(* CoDeSys 2.3.9.55 project: coolingskidlogic.pro *)
(* Libraries: Standard.lib 20.5.14 01:13:26, Iecsfc.lib 30.1.13 06:05:12, SYSLIBCALLBACK.LIB 30.1.13 06:05:12 *)

(* PLC configuration (modules and I/O channels)
xWaterLow AT %IX10.0 [BOOLOnX_I] Ch_1 Digital input
xWaterLowLow AT %IX10.1 [BOOLOnX_I] Ch_2 Digital input
AT %IX10.2 [BOOLOnX_I] Ch_1 Digital input
AT %IX10.3 [BOOLOnX_I] Ch_2 Digital input
AT %IX10.4 [BOOLOnX_I] Ch_3 Digital input
AT %IX10.5 [BOOLOnX_I] Ch_4 Digital input
0750-0402 4 DI 24 V DC 3.0ms [Type_1_4_Channels] node 2, in %IX10.2 out %QB4
  AT %IX10.6 [BOOLOnX_I] Ch_1 Digital input
  AT %IX10.7 [BOOLOnX_I] Ch_2 Digital input
  AT %IX10.8 [BOOLOnX_I] Ch_3 Digital input
  AT %IX10.9 [BOOLOnX_I] Ch_4 Digital input
xOutput8DO1 AT %QX2.0 [BOOLOnX_Q] Ch_1 Digital output
AT %QX2.1 [BOOLOnX_Q] Ch_2 Digital output
AT %QX2.2 [BOOLOnX_Q] Ch_3 Digital output
AT %QX2.3 [BOOLOnX_Q] Ch_4 Digital output
AT %QX2.4 [BOOLOnX_Q] Ch_5 Digital output
AT %QX2.5 [BOOLOnX_Q] Ch_6 Digital output
AT %QX2.6 [BOOLOnX_Q] Ch_7 Digital output
AT %QX2.7 [BOOLOnX_Q] Ch_8 Digital output
xOutput AT %QX2.8 [BOOLOnX_Q] Ch_1 Digital output
AT %QX2.9 [BOOLOnX_Q] Ch_2 Digital output
AT %QX2.10 [BOOLOnX_Q] Ch_1 Digital output
AT %QX2.11 [BOOLOnX_Q] Ch_2 Digital output
0750-0492 2 AI 4-20mA Diff Measurement Input [Type_8_2_Channels] node 6, in %IB20 out %QB0
  AT %IW0 [WORDOnW_I] Ch_1 Input word
  AT %IW1 [WORDOnW_I] Ch_2 Input word
0750-0461 2 AI PT100 (RTD) [Type_44_2_Channels] node 7, in %IB20 out %QB0
  AT %IW2 [INTOnW_I] Ch_1 signed Input value
  AT %IW3 [INTOnW_I] Ch_2 signed Input value
0750-0461 2 AI PT100 (RTD) [Type_44_2_Channels] node 8, in %IB24 out %QB0
  AT %IW4 [INTOnW_I] Ch_1 signed Input value
  AT %IW5 [INTOnW_I] Ch_2 signed Input value
0750-0455 4 AI 4-20mA s.e. [Type_8_4_Channels] node 9, in %IB28 out %QB0
  AT %IW6 [WORDOnW_I] Ch_1 Input word
  AT %IW7 [WORDOnW_I] Ch_2 Input word
  AT %IW8 [WORDOnW_I] Ch_3 Input word
  AT %IW9 [WORDOnW_I] Ch_4 Input word
0750-0554 2 AO 4-20mA [Type_14_2_Channels] node 10, in %IB32 out %QB0
  AT %QW0 [WORDOnW_Q] Ch_1 Analog output
  AT %QW1 [WORDOnW_Q] Ch_2 Analog output
AT %IX10.10 [BOOLOnX_I] Ch_1 Digital input
AT %IX10.11 [BOOLOnX_I] Ch_2 Digital input
AT %IX10.12 [BOOLOnX_I] Ch_3 Digital input
AT %IX10.13 [BOOLOnX_I] Ch_4 Digital input
Modbus variables [PFC200MODBUS] node 1, in %IB0 out %QB0 {PlcStopBehaviour = 1; FiledbusErrorBehaviour = 1; TcpOperation = 1; TcpPort = 502; TcpTimeout = 600; UdpOperation = 1; UdpPort = 502; RtuOperation = 0; NodeId = 1; ResponseTimeout = 100; Interface = 0; Baud = 115200; StopBits = 1; Parity = 1; FlowCtrl = 0; PhysInterface = 0}
Modbus-Master [MB_MASTER] node 2, in %IB0 out %QB0
*)

(* Global variable list: Global_Variables *)
VAR_GLOBAL
	gaPumps: ARRAY [1..2] OF  ST_PUMP;
	gaTemps: ARRAY [1..3] OF ST_RTD;
	gaSwitches: ARRAY [1..3] OF ST_SWITCH;
	gaFans: ARRAY [1..4] OF ST_FAN;
	gConductivity: ST_COND;
	gFlow: ST_FLOW;
	gAct: ST_ACT;
	gSystem: ST_SYSTEM;
	gcAlarm: INT :=  1;
	gcFault:  INT := 0;
	gTempValCtrlSys: ST_TempValCtrlSys;
	gProgramErrors: ST_ProgramErrors;
	tbFailure: BOOL;
	tbSuccess: BOOL;
	tbTBLog: STRING(256);

	activePump: ST_PUMP;
	standbyPump: ST_PUMP;


END_VAR

(* Data type in Legacy *)
TYPE BAD :
STRUCT
END_STRUCT
END_TYPE

(* Data type in Legacy *)
TYPE HERE :
STRUCT
	On: BOOL;
	Off: BOOL;
	Fault: BOOL;
	Shutting_Down: BOOL;
	Initializing: BOOL;
	Calibrating: BOOL;
	Acknowledge_Fault: BOOL;
	LIST_FLAGS: ARRAY [1..25] OF BOOL;
	System_Active: BOOL;
	ManualRequest: BOOL;
	AutoRequest: BOOL;
	BAD_Duplex: BOOL;
	ALERT_Simplex: BOOL;
	REQ_Switch: BOOL;
	ALERT_PriActive: BOOL;
	ALERT_SecActive: BOOL;
END_STRUCT
END_TYPE

(* Data type in Instrument Data Types *)
TYPE RAWINPUT :
STRUCT
	wRawAnalogWord: WORD;
	iRawAnalogInt: INT;
	xRawDigital: BOOL;
END_STRUCT
END_TYPE

(* Data type in Legacy *)
TYPE SignalIO :
STRUCT
END_STRUCT
END_TYPE

(* Data type in Legacy *)
TYPE ST_ACT :
STRUCT
	stDescription: ST_Description;
	stActualization: ST_Analog;
	stCounters: ST_LGCount;
	stCalibrationStatus: ST_CalTest;
	rOpenPerc: REAL; (*Percentage of it being Open*)
END_STRUCT
END_TYPE

(* Data type in Legacy *)
TYPE ST_ActivePumpStandbyPump :
STRUCT
END_STRUCT
END_TYPE

(* Data type in Legacy *)
TYPE ST_Analog :
STRUCT
	rGain: REAL;
	rOffset: REAL;
	iRaw: REAL;
	rProcessed: REAL;
END_STRUCT
END_TYPE

(* Data type in Legacy *)
TYPE ST_Backup :
STRUCT
	xActive: BOOL;
	xRedundant: BOOL;
END_STRUCT
END_TYPE

(* Data type in Legacy *)
TYPE ST_CalTest :
STRUCT
	xCalibrated: BOOL;
	xTested: BOOL;
END_STRUCT
END_TYPE

(* Data type in Legacy *)
TYPE ST_COND :
STRUCT
	stDescription: ST_Description;
	stConductivity: ST_Analog; (*Cond Reading Power*)
	stFault: ST_Digital; (*Fault Y/N*)
	stAlarm: ST_DIgital; (*Alarm Y/N*)
	stCounters: ST_LGCount;
	stCalibrationStatus: ST_CalTest;
END_STRUCT
END_TYPE

(* Data type in Legacy *)
TYPE ST_Count :
STRUCT
	iAlarm: INT;
	iFault: INT;
	iForce: INT;
	iCalibrate: INT;
	iTest: INT;
END_STRUCT
END_TYPE

(* Data type in Instrument Data Types *)
TYPE ST_DC :
STRUCT
	arRealValues: ARRAY [1..10] OF REAL;
	axBoolValues: ARRAY [1..10] OF BOOL;
	aiIntValues: ARRAY [1..10] OF INT;
	awWordValues: ARRAY [1..10] OF WORD;
END_STRUCT
END_TYPE

(* Data type in Legacy *)
TYPE ST_Description :
STRUCT
	iID : INT;
	iState: INT; (*Offline, Standby,  Active, Calibration, Testing *)
	xFault: BOOL;
	xAlarm: BOOL;
	sDetail:  STRING;
END_STRUCT
END_TYPE

(* Data type in Legacy *)
TYPE ST_Digital :
STRUCT
	iValue: INT;
END_STRUCT
END_TYPE

(* Data type in Legacy *)
TYPE ST_FA :
STRUCT
	xFault: BOOL;
	xAlarm: BOOL;
END_STRUCT
END_TYPE

(* Data type in Legacy *)
TYPE ST_FAN :
STRUCT
	stDescription: ST_Description;
	stActivate: ST_Digital; (*Pump On/Off*)
	stCounters: ST_LGCount;
	stCalibrationStatus: ST_CalTest;
	stBackup: ST_Backup;
END_STRUCT
END_TYPE

(* Data type in Legacy *)
TYPE ST_FLOW :
STRUCT
	stDescription: ST_Description;
	stFlowRate: ST_Analog; (*Switch Trip*)
	stCounters: ST_LGCount;
	stCalibrationStatus: ST_CalTest;
END_STRUCT
END_TYPE

(* Data type in Legacy *)
TYPE ST_HeartBeat :
STRUCT
	stDescription: ST_Description;
END_STRUCT
END_TYPE

(* Data type in Instrument Data Types *)
TYPE ST_INSTRUMENT :
STRUCT
	iState: INT; (*0 = Standby; 1 = Data Loading;*)
	stInput: ST_IO;
	stOutput: ST_IO;
	stMeasurement: ST_MEASUREMENTS;
	stActuateValues: ST_MEASUREMENTS;
END_STRUCT
END_TYPE

(* Data type in Flags *)
TYPE ST_InstrumentFlags :
STRUCT
	xConductivitySensorAlarmTrip: BOOL := FALSE;
	xConductivitySensorFaultTrip: BOOL := FALSE;
	xPump1BadRead: BOOL := FALSE;
	xPump2BadRead: BOOL := FALSE;
	xPump1LPError: BOOL := FALSE;
	xPump2LPError: BOOL := FALSE;
	xConductivitySensorBadRead: BOOL := FALSE;
	xConductivitySensorMisalignment: BOOL := FALSE;
	xConductivitySensorError: BOOL := FALSE;
	xFlowSensorBadRead: BOOL := FALSE;
	xRTD1BadRead: BOOL := FALSE;
	xRTD2BadRead: BOOL := FALSE;
	xRTD3BadRead: BOOL := FALSE;
	xNoPumpBackup: BOOL := FALSE;
	xPump1Failure: BOOL := FALSE;
	xPump2Failure: BOOL := FALSE;
	xRTD1Failure: BOOL := FALSE;
	xRTD2Failure: BOOL := FALSE;
	xRTD3Failure: BOOL := FALSE;
	xConductivitySensorFailure: BOOL := FALSE;
	xFlowSensorFailure: BOOL := FALSE;
	xPressureLow: BOOL := FALSE;
	xPumpPowerLow: BOOL := FALSE;
	xFlowLow: BOOL := FALSE;
	xWaterLevelSensorError: BOOL := FALSE;
END_STRUCT
END_TYPE

(* Data type in Legacy *)
TYPE ST_IO :
STRUCT
	axDigital: ARRAY [1..100] OF BOOL;
	awAnalog: ARRAY[1..100] OF WORD;
	aiAnalog: ARRAY[1..100] OF INT;
END_STRUCT
END_TYPE

(* Data type in Legacy *)
TYPE ST_LGCount :
STRUCT
	stLocal : ST_Count;
	stGlobal: ST_Count;
END_STRUCT
END_TYPE

(* Data type in Instrument Data Types *)
TYPE ST_MEASUREMENTS :
STRUCT
	axDigital: ARRAY [1..100] OF BOOL;
	arAnalog: ARRAY[1..100] OF REAL;
END_STRUCT
END_TYPE

(* Data type in Legacy *)
TYPE ST_PRES :
STRUCT
	stDescription: ST_Description;
	stSwitchTrip: ST_Digital; (*Switch Trip*)
	stCounters: ST_LGCount;
	stCalibrationStatus: ST_CalTest;
END_STRUCT
END_TYPE

(* Data type in Legacy *)
TYPE ST_ProgramErrors :
STRUCT
	xTempValCtrlSys: BOOL;
	xDataConversion: BOOL;
END_STRUCT
END_TYPE

(* Data type in Legacy *)
TYPE ST_PUMP :
STRUCT
	stDescription: ST_Description;
	stPumpPower: ST_Analog; (*Pump Power*)
	stActivate: ST_Digital; (*Pump On/Off*)
	stCounters: ST_LGCount;
	stCalibrationStatus: ST_CalTest;
	stBackup: ST_Backup;
END_STRUCT
END_TYPE

(* Data type in Legacy *)
TYPE ST_RTD :
STRUCT
	stDescription: ST_Description;
	stTempRead: ST_Analog;
	stCounters: ST_LGCount;
	stCalibrationStatus: ST_CalTest;
END_STRUCT
END_TYPE

(* Data type in Legacy *)
TYPE ST_SPT :
STRUCT
	rSetpoint: REAL;
	rThreshold: REAL;
END_STRUCT
END_TYPE

(* Data type in Legacy *)
TYPE ST_SWITCH :
STRUCT
	stDescription: ST_Description;
	stSwitchTrip: ST_Digital; (*Switch Trip*)
	stCounters: ST_LGCount;
	stCalibrationStatus: ST_CalTest;
END_STRUCT
END_TYPE

(* Data type in Legacy *)
TYPE ST_SYSTEM :
STRUCT
	stSystemCounters: ST_SystemCounters;
	stSystemFlags: ST_SystemFlags;
	stInstrumentFlags: ST_instrumentFlags;
	stInputs: ST_SystemInputs;
	stOutputs: ST_SystemOutputs;
END_STRUCT
END_TYPE

(* Data type in Legacy *)
TYPE ST_SystemCounters :
STRUCT
	iRTDFailures: INT;
	iPumpFailures: INT;
	iActivePump: INT;
	iActiveFanGroup: INT;
END_STRUCT
END_TYPE

(* Data type in Legacy *)
TYPE ST_SystemFlags :
STRUCT
	xSwitchPumpRequest: BOOL;
	xAwaitInitialization: BOOL;
	xAwaitCalibration: BOOL;
	xFault: BOOL;
	xAlarm: BOOL;
	xPPFError: BOOL;
	xWaterLow: BOOL;
	xWaterVeryLow: BOOL;
END_STRUCT
END_TYPE

(* Data type in Legacy *)
TYPE ST_SystemInputs :
STRUCT
	rPumpPower: REAL;
	rFlowRate: REAL;
	rConductivity: REAL;
	rTemperature: REAL;
	xPressureLow: BOOL;
	xWaterLow: BOOL;
	xWaterLowLow: BOOL;
	xSystemON: BOOL;
	xConductivityAlarm: BOOL;
	xConductivityFault: BOOL;
END_STRUCT
END_TYPE

(* Data type in Legacy *)
TYPE ST_SystemMeasurement :
STRUCT

END_STRUCT
END_TYPE

(* Data type in Legacy *)
TYPE ST_SystemOutputs :
STRUCT
	rValveActuate: REAL;
	xPump1Activate: BOOL;
	xPump2Activate: BOOL;
	xFan12Activate: BOOL;
	xFan34Activate: BOOL;
END_STRUCT
END_TYPE

(* Data type in Legacy *)
TYPE ST_TempValCtrlSys :
STRUCT
	rDiffThresh: REAL;
	rDiffTol: REAL;
	iSysMeasState: INT;
	xFault: BOOL; (*Fault when all controlers are bad, or program error*)
	xAlarm: BOOL; (*Alarm for fault, when controller is bad, or program error*)
END_STRUCT
END_TYPE

(* POU PLC_PRG, LD *)
PROGRAM PLC_PRG
VAR PERSISTENT
	stPump1: ST_INSTRUMENT;
	stPump2: ST_INSTRUMENT;
	stPump3: ST_INSTRUMENT;
	stRTD1: ST_INSTRUMENT;
	stRTD2: ST_INSTRUMENT;
	stRTD3: ST_INSTRUMENT;
	stFan1: ST_INSTRUMENT;
	stFan2: ST_INSTRUMENT;
	stFan3: ST_INSTRUMENT;
	stFan4: ST_INSTRUMENT;
	stConductivitySensor: ST_INSTRUMENT;
	stFlowSensor: ST_INSTRUMENT;
	stWaterLevelLow: ST_INSTRUMENT;
	stWaterLevelLowLow: ST_INSTRUMENT;
	stPressureLowSensor: ST_INSTRUMENT;
	stSystemRunSwitch: ST_INSTRUMENT;

	stInstrumentFlags: ST_InstrumentFlags;

	stSystem: ST_SYSTEM;
END_VAR
VAR
		xReadAnalog: BOOL;
	xReadTemperature: BOOL;
	fbRunTestBench: RunTestBench;
	xTesting: BOOL;
	xReadDigital: BOOL;
	fbWaterLevelLowCaputer: FB_DigitalCapture;
	fbWaterLevelLowLowCapture: FB_DigitalCapture;
	fbConductivityAlarmCapture: FB_DigitalCapture;
	fbAssignAnalogValues: FB_AssignAnalog;
	fbAAP1: FB_AssignAnalog;
	fbAAP2: FB_AssignAnalog;
	fbAARTD1: FB_AssignAnalog;
	fbAARTD2: FB_AssignAnalog;
	fbAARTD3: FB_AssignAnalog;
	fbAAF3: FB_AssignAnalog;
	fbAAF: FB_AssignAnalog;
	fbAAC: FB_AssignAnalog;
END_VAR
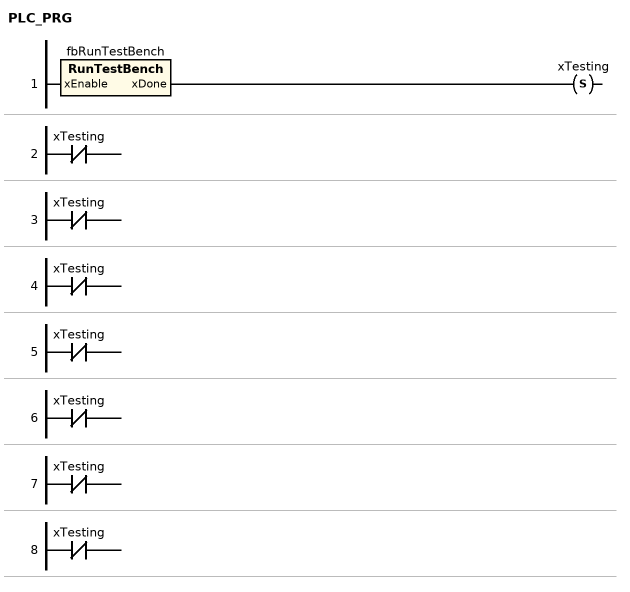
_LD_ (* Ladder Diagram *)
NETWORK 1
	fbRunTestBench:RunTestBench(xEnable: *) --- (S xTesting)
NETWORK 2
	[/xTesting]
NETWORK 3
	[/xTesting]
NETWORK 4
	[/xTesting]
NETWORK 5
	[/xTesting]
NETWORK 6
	[/xTesting]
NETWORK 7
	[/xTesting]
NETWORK 8
	[/xTesting]
_END_LD_
(* the same logic as Structured Text *)
(* Network 1 *)
fbRunTestBench(xEnable := TRUE);
IF fbRunTestBench.xDone THEN xTesting := TRUE; END_IF;
(* Network 2 *)
(* Network 3 *)
(* Network 4 *)
(* Network 5 *)
(* Network 6 *)
(* Network 7 *)
(* Network 8 *)
END_PROGRAM

(* POU RunTestBench, ST *)
FUNCTION_BLOCK RunTestBench
VAR_INPUT
	xEnable: BOOL;
END_VAR
VAR_OUTPUT
	xDone: BOOL := TRUE;
END_VAR
VAR
	istopCase: INT;
	iWait: INT := 0;
END_VAR
IF xEnable = FALSE THEN
	RETURN;
END_IF
TB_MainProgram2();
END_FUNCTION_BLOCK

(* POU TB_MainProgram2, LD *)
PROGRAM TB_MainProgram2
VAR
	dummywordsignals: ARRAY [1..4] OF WORD :=
	5000,
	6000,
	4000,
	3000;
	dummyintsignals: ARRAY[1..3] OF INT :=
	4100,
	4100,
	4100;
	dummyboolsignals: ARRAY[1..5] OF BOOL :=
	FALSE,
	FALSE,
	FALSE,
	FALSE,
	FALSE;


	arInputNormBounds: ARRAY [1..14] OF REAL :=
	10000, (*Primary Pump Max Signal*)
	10000, (*Secondary  Pump Max Signal*)
	10000, (*RTD 1 Max Signal*)
	10000, (*RTD 2 Max Signal*)
	10000, (*RTD 3 Max Signal*)
	10000, (*Conductivity Sensor  Max Signal*)
	10000, (*Flow  Sensor  Max Signal*)
	0, (*Primary Pump Min Signal *)
	0 , (*Secondary Pump Min Signal *)
	0, (*RTD 1 Min Signal *)
	0, (*RTD 2 Min Signal *)
	0, (*RTD 3 Min Signal *)
	0, (*Conductivity Sensor  Min Signal *)
	0; (*Flow Sensor  Min Signal *)
	arInputNormTol: ARRAY [1..7] OF REAL :=
	0.1, (*Primary Pump Normalized Signal Tolerance*)
	0.1, (*Secondary  Pump Normalized Signal Tolerance*)
	0.1, (*RTD 1 Max Normalized Signal Tolerance*)
	0.1, (*RTD 2 Max Normalized Signal Tolerance*)
	0.1, (*RTD 3 Max Normalized Signal Tolerance*)
	0.1, (*Conductivity Sensor  Normalized Signal Tolerance*)
	0.1; (*Flow  Sensor  Normalized Signal Tolerance*)
	arInputValBounds: ARRAY [1..14] OF REAL :=
	100, (*Primary Pump Max Value*)
	100, (*Secondary  Pump Max Value*)
	100, (*RTD 1 Max Value*)
	100, (*RTD 2 Max Value*)
	100, (*RTD 3 Max Value*)
	100, (*Conductivity Sensor  Max Value*)
	100, (*Flow  Sensor  Max Value*)
	0, (*Primary Pump Min Value *)
	0 , (*Secondary Pump Min Value *)
	0, (*RTD 1 Min Value *)
	0, (*RTD 2 Min Value *)
	0, (*RTD 3 Min Value *)
	0, (*Conductivity Sensor  Min Value *)
	0; (*Flow Sensor  Min Value *)



	awWordInputSignal: ARRAY [1..4] OF WORD; (*Primary Pump, Secondary Pump, Conductivity, Flow*)
	aiIntInputSignal: ARRAY [1..3] OF INT; (*RTD 1, RTD 2, RTD 3*)

	arNormInputSignals: ARRAY [1..7] OF REAL; (*Primary Pump, Secondary Pump, RTD 1, RTD 2, RTD 3, Conductivity, Flow*)
	axBoolDebouncedInputSignal: ARRAY [1..5] OF BOOL; (*Water Level Low, Water Level Low Low,  Low Pressure, Conductivity Alarm, Conductivity Fault  *)
	arMultiSignals: ARRAY [1..5] OF REAL; (*Primary Pump, Secondary Pump, RTD 1, RTD 2, RTD 3*)

	arLinearizedInputSignals: ARRAY [1..4] OF REAL; (*Pump Power, Temperature, Conductivity, Flow*)
	axBoolInputSignal: ARRAY [1..5] OF BOOL; (*Water Level Low, Water Level Low Low, Pressure, Conductivity Alarm, Conductivity Fault *)

	emptyIntSignals: ARRAY [1..10] OF INT;
	emptyWordSignals: ARRAY [1..10] OF WORD;


	axInputSignalFlags: ARRAY [1..5] OF BOOL; (*1. Bad Primary Pump Signal,  2. Bad Secondary Pump Signal,  3. Bad RTD 1 Signal, 4. Bad RTD 2 Signal,  5.Bad RTD 3 Signal*)
	axFaultFlags: ARRAY[1..25] OF BOOL; (*1. Bad Conductivity Signal,  2. Bad Flow Signal, 3. Duplex Failure, 4. Critical Vessel Level , 5. Bad Level Signal 6. Conductivity Sensor Malfunction 7. Critical Coolant Conductivity 8. Critical Coolant Temperature*)
	axAutoTurnoverRequests: ARRAY[1..2] OF BOOL;
	axActivePumps: ARRAY[1..2] OF BOOL; (*Primary Pump Active, Secondary Pump Active*)
	axActiveFans: ARRAY [1..2] OF BOOL; (*Primary Fan Active, Secondary Fan Active*)
	axSystemAlerts: ARRAY [1..20] OF BOOL; (*1 On, 2 Shutting Down,3  Initializing, 4 calibrating,  5 simplex mode,  6. Low Vessel Level , 7. High Coolant Conductivity 8. Low Pump Power 9. Low Hydraulic Flow 10. Low Hydraulic Pressure, 11. Coolant Temperature Warning, 12. Fan 1 Overide 13. Fan 2 Control Overide14. Force Throughput 15. Manually Control Thruput 16. Fans Auto Enabled 17. Manually Control Fans*)

	axHydraulicFailures: ARRAY [1..2] OF BOOL; (*Primary Hydraulic Failure 2. Secondary Hydraulic Failure*)


	iBadRTDs: INT;

	USERMasterStart: BOOL;
	USERAcknowledgeFault: BOOL;
	USERShutdown: BOOL;
	USERTurnoverRequest: BOOL;
	xMasterAutoTurnoverRequest: BOOL;
	xMasterTurnoverRequest: BOOL;
	xMasterFault: BOOL;

	rPercentValveOpen: REAL;
	fbcheckwaterlevel: FB_CheckWaterLevel;
	fbcheckconductivity: FB_CheckConductivity;
	fbpowerpressureflowthreshold: FB_PowerPressureFlowThreshold;
	fbpowerpressureflowvote: FB_PowerPressureFlowVote;
	fbtempboundcheck: FB_TemperatureBoundCheck;
	fbsysstart: FB_SystemStart;
	fbfaultcheck: FB_FaultCheck;
	fbstop: FB_SystemStop;
	fbpsc: FB_PumpSwitchControl;
	fbpc: FB_PumpControl;
	fbsil: FB_SwitchInitLink;
	fbpump1assign: FB_AssignAnalog;
	fbpump2assign: FB_AssignAnalog;
	fbrtd1assign: FB_AssignAnalog;
	fbrtd2assign: FB_AssignAnalog;
	fbrtd3assign: FB_AssignAnalog;
	fbcondassign: FB_AssignAnalog;
	fbflowassign: FB_AssignAnalog;
	fbwaterlevellow: FB_AssignDigital;
	fbwaterlevellowlowlow: FB_AssignDigital;
	fbpvv: FB_PumpValueValidation;
	fbtsa: FB_TempSystemAlignment;
	fbcondwarning: FB_AssignDigital;
	fbcondfault: FB_AssignDigital;
	fbmatl: FB_MasterAutoTurnoverLink;
	fbfc: FB_FanControl;
	fbtc: FB_TemperatureController;
	fbpressure: FB_AssignDigital;
	fbtcoo: FB_TemperatureControllerOnOff;
END_VAR
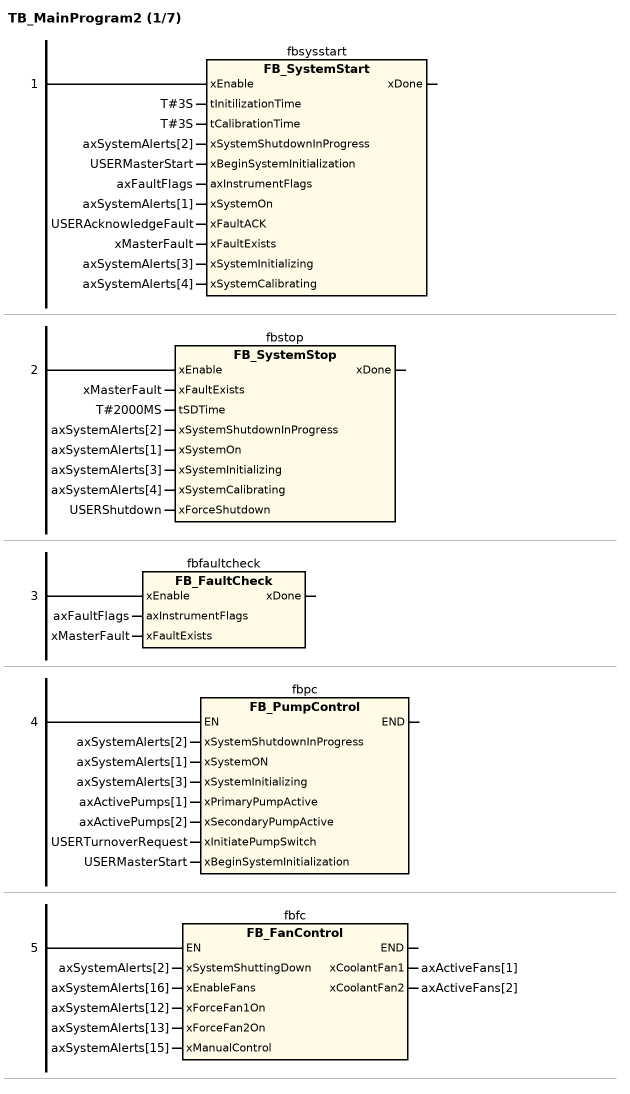
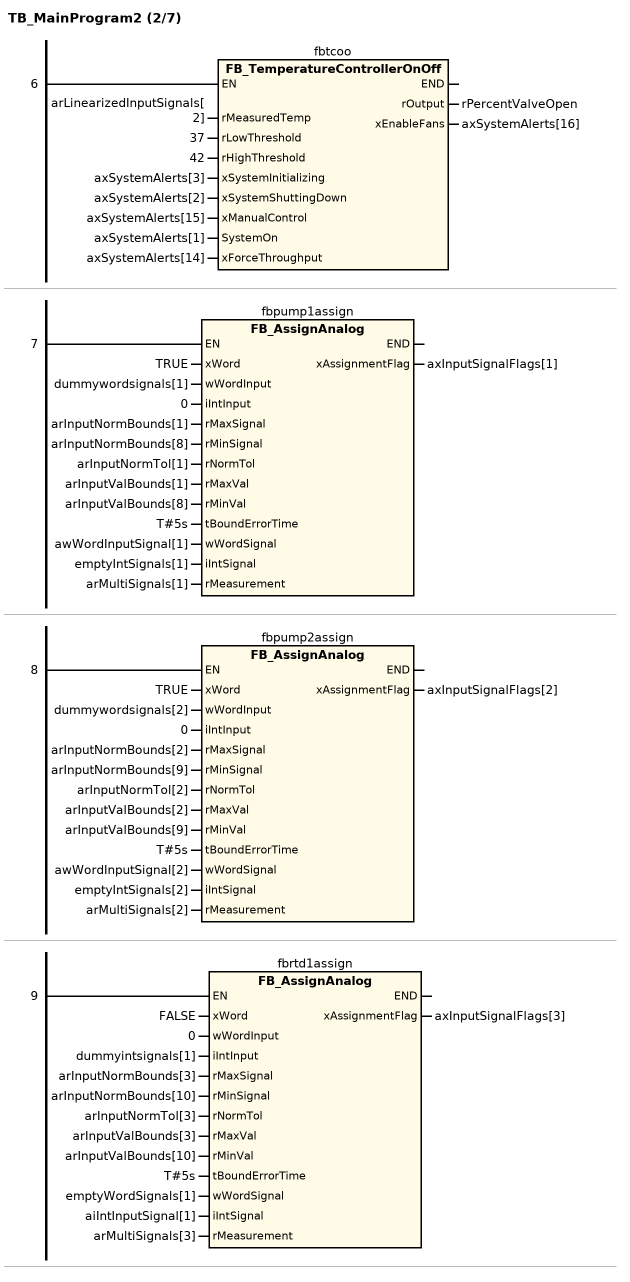
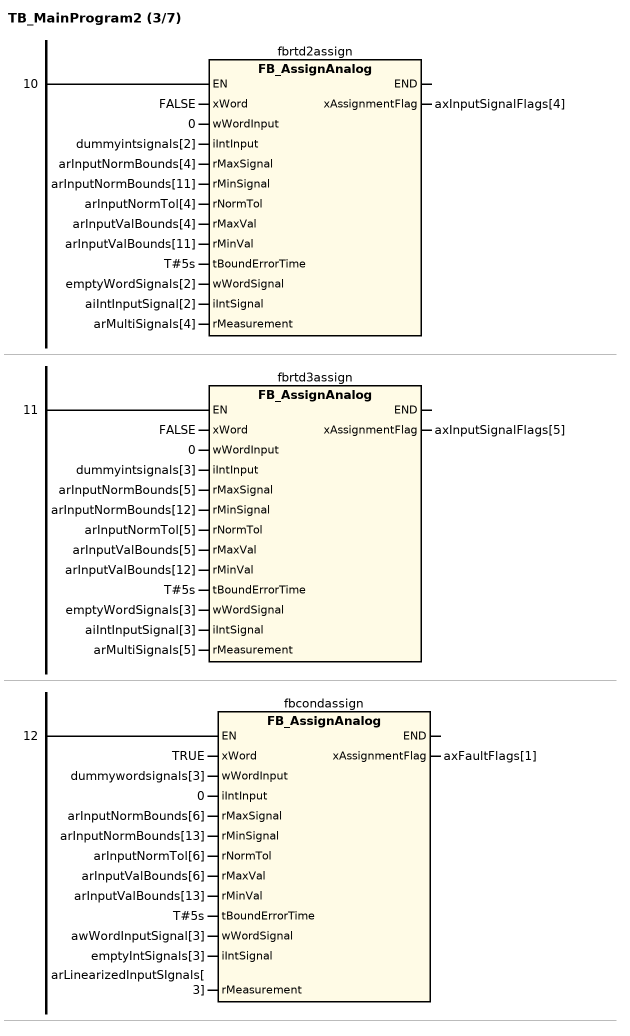
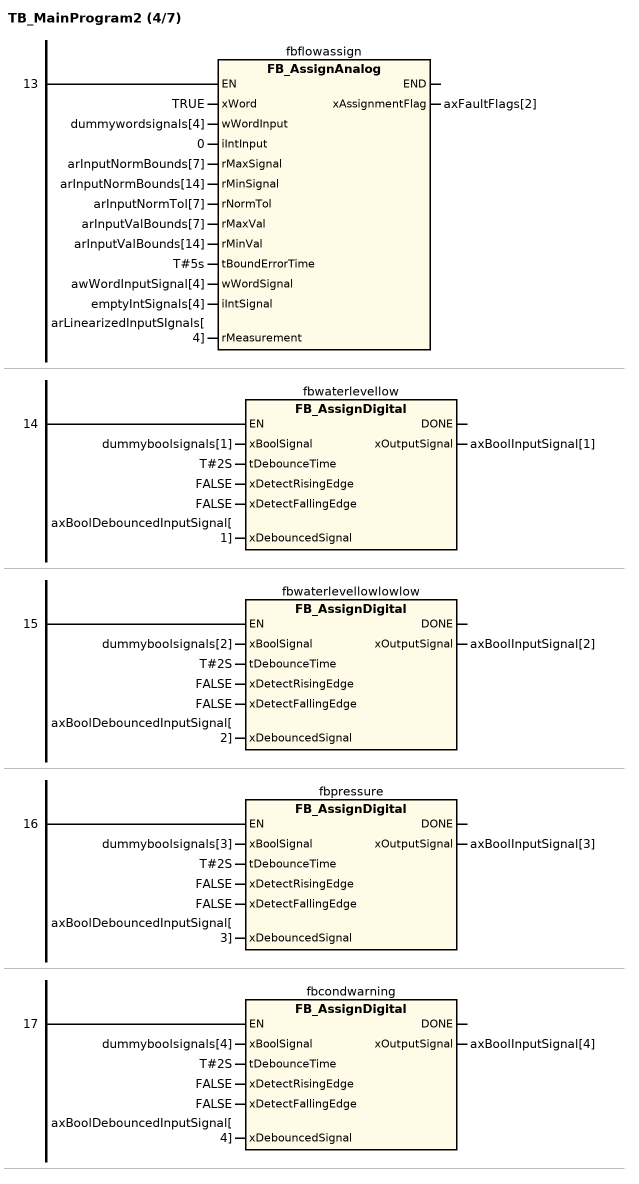
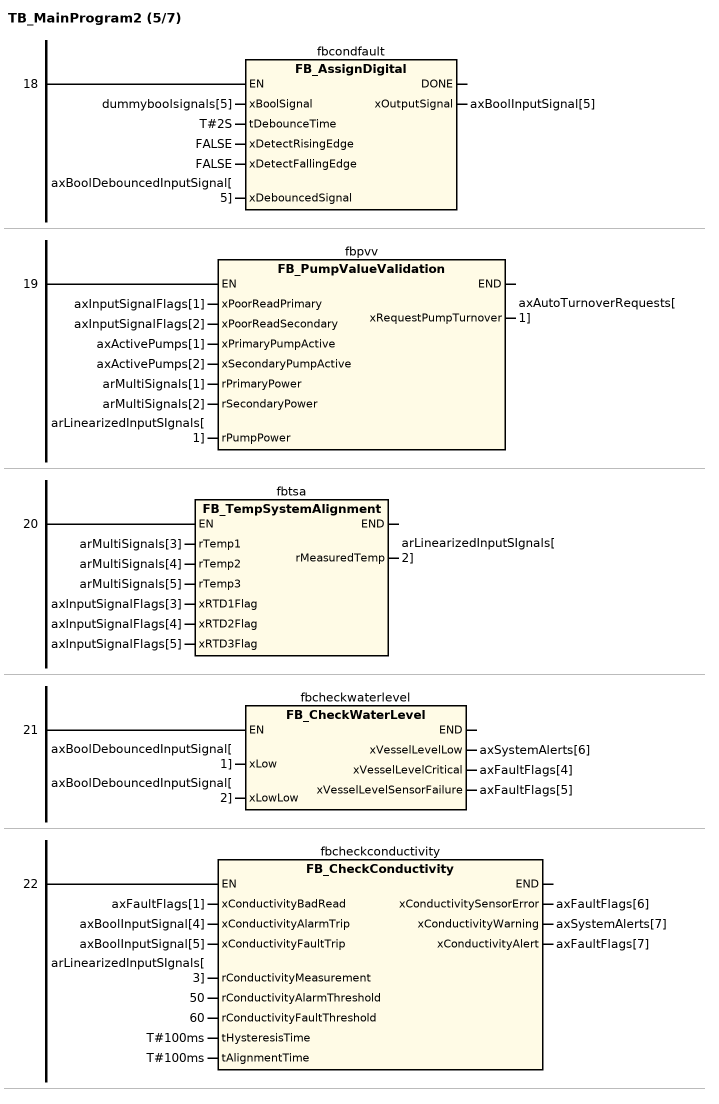
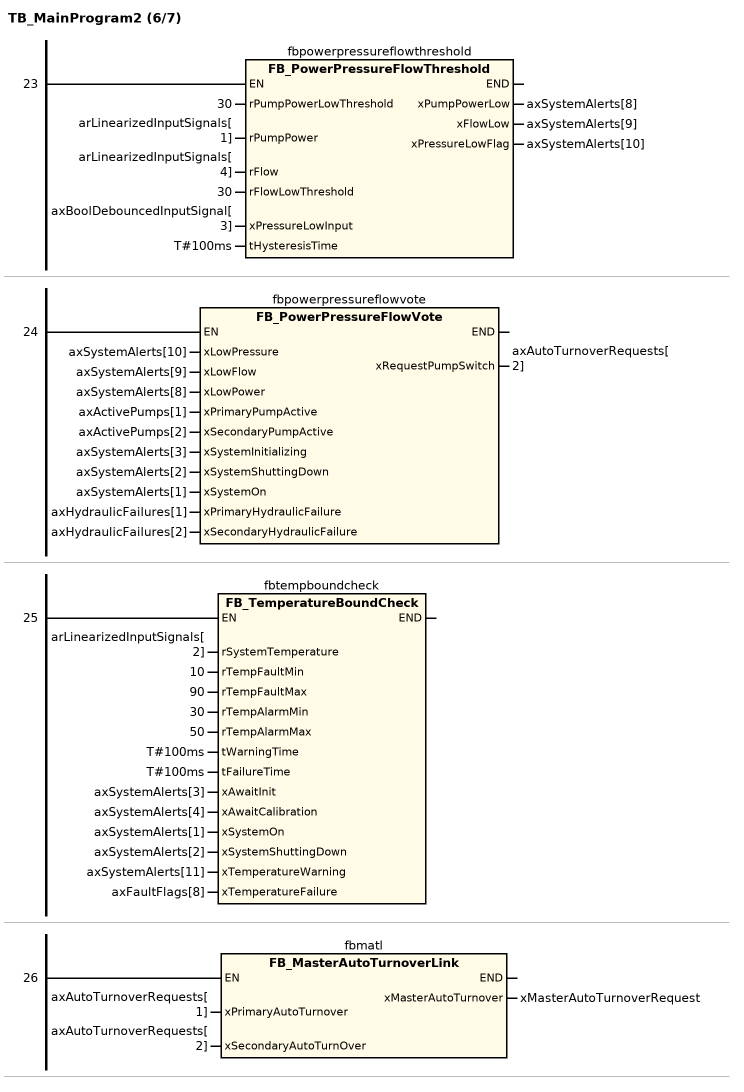
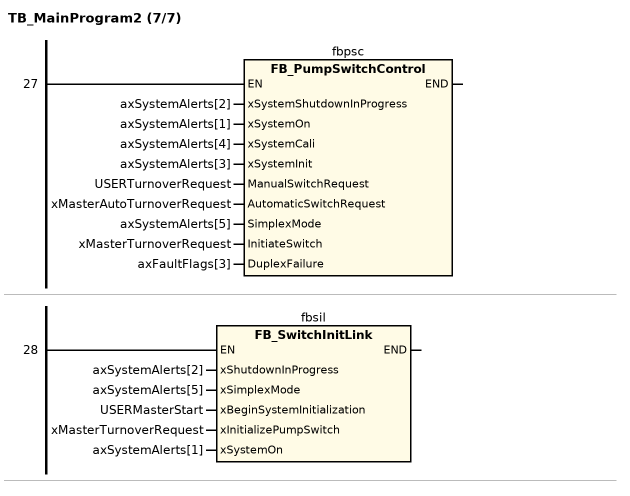
_LD_ (* Ladder Diagram *)
NETWORK 1
	fbsysstart:FB_SystemStart(xEnable: *, tInitilizationTime: T#3S, tCalibrationTime: T#3S, xSystemShutdownInProgress: axSystemAlerts[2], xBeginSystemInitialization: USERMasterStart, axInstrumentFlags: axFaultFlags, xSystemOn: axSystemAlerts[1], xFaultACK: USERAcknowledgeFault, xFaultExists: xMasterFault, xSystemInitializing: axSystemAlerts[3], xSystemCalibrating: axSystemAlerts[4])
NETWORK 2
	fbstop:FB_SystemStop(xEnable: *, xFaultExists: xMasterFault, tSDTime: T#2000MS, xSystemShutdownInProgress: axSystemAlerts[2], xSystemOn: axSystemAlerts[1], xSystemInitializing: axSystemAlerts[3], xSystemCalibrating: axSystemAlerts[4], xForceShutdown: USERShutdown)
NETWORK 3
	fbfaultcheck:FB_FaultCheck(xEnable: *, axInstrumentFlags: axFaultFlags, xFaultExists: xMasterFault)
NETWORK 4
	fbpc:FB_PumpControl(EN: *, xSystemShutdownInProgress: axSystemAlerts[2], xSystemON: axSystemAlerts[1], xSystemInitializing: axSystemAlerts[3], xPrimaryPumpActive: axActivePumps[1], xSecondaryPumpActive: axActivePumps[2], xInitiatePumpSwitch: USERTurnoverRequest, xBeginSystemInitialization: USERMasterStart)
NETWORK 5
	fbfc:FB_FanControl(EN: *, xSystemShuttingDown: axSystemAlerts[2], xEnableFans: axSystemAlerts[16], xForceFan1On: axSystemAlerts[12], xForceFan2On: axSystemAlerts[13], xManualControl: axSystemAlerts[15], xCoolantFan1 => axActiveFans[1], xCoolantFan2 => axActiveFans[2])
NETWORK 6
	fbtcoo:FB_TemperatureControllerOnOff(EN: *, rMeasuredTemp: arLinearizedInputSignals[2], rLowThreshold: 37, rHighThreshold: 42, xSystemInitializing: axSystemAlerts[3], xSystemShuttingDown: axSystemAlerts[2], xManualControl: axSystemAlerts[15], SystemOn: axSystemAlerts[1], xForceThroughput: axSystemAlerts[14], rOutput => rPercentValveOpen, xEnableFans => axSystemAlerts[16])
NETWORK 7
	fbpump1assign:FB_AssignAnalog(EN: *, xWord: TRUE, wWordInput: dummywordsignals[1], iIntInput: 0, rMaxSignal: arInputNormBounds[1], rMinSignal: arInputNormBounds[8], rNormTol: arInputNormTol[1], rMaxVal: arInputValBounds[1], rMinVal: arInputValBounds[8], tBoundErrorTime: T#5s, wWordSignal: awWordInputSignal[1], iIntSignal: emptyIntSignals[1], rMeasurement: arMultiSignals[1], xAssignmentFlag => axInputSignalFlags[1])
NETWORK 8
	fbpump2assign:FB_AssignAnalog(EN: *, xWord: TRUE, wWordInput: dummywordsignals[2], iIntInput: 0, rMaxSignal: arInputNormBounds[2], rMinSignal: arInputNormBounds[9], rNormTol: arInputNormTol[2], rMaxVal: arInputValBounds[2], rMinVal: arInputValBounds[9], tBoundErrorTime: T#5s, wWordSignal: awWordInputSignal[2], iIntSignal: emptyIntSignals[2], rMeasurement: arMultiSignals[2], xAssignmentFlag => axInputSignalFlags[2])
NETWORK 9
	fbrtd1assign:FB_AssignAnalog(EN: *, xWord: FALSE, wWordInput: 0, iIntInput: dummyintsignals[1], rMaxSignal: arInputNormBounds[3], rMinSignal: arInputNormBounds[10], rNormTol: arInputNormTol[3], rMaxVal: arInputValBounds[3], rMinVal: arInputValBounds[10], tBoundErrorTime: T#5s, wWordSignal: emptyWordSignals[1], iIntSignal: aiIntInputSignal[1], rMeasurement: arMultiSignals[3], xAssignmentFlag => axInputSignalFlags[3])
NETWORK 10
	fbrtd2assign:FB_AssignAnalog(EN: *, xWord: FALSE, wWordInput: 0, iIntInput: dummyintsignals[2], rMaxSignal: arInputNormBounds[4], rMinSignal: arInputNormBounds[11], rNormTol: arInputNormTol[4], rMaxVal: arInputValBounds[4], rMinVal: arInputValBounds[11], tBoundErrorTime: T#5s, wWordSignal: emptyWordSignals[2], iIntSignal: aiIntInputSignal[2], rMeasurement: arMultiSignals[4], xAssignmentFlag => axInputSignalFlags[4])
NETWORK 11
	fbrtd3assign:FB_AssignAnalog(EN: *, xWord: FALSE, wWordInput: 0, iIntInput: dummyintsignals[3], rMaxSignal: arInputNormBounds[5], rMinSignal: arInputNormBounds[12], rNormTol: arInputNormTol[5], rMaxVal: arInputValBounds[5], rMinVal: arInputValBounds[12], tBoundErrorTime: T#5s, wWordSignal: emptyWordSignals[3], iIntSignal: aiIntInputSignal[3], rMeasurement: arMultiSignals[5], xAssignmentFlag => axInputSignalFlags[5])
NETWORK 12
	fbcondassign:FB_AssignAnalog(EN: *, xWord: TRUE, wWordInput: dummywordsignals[3], iIntInput: 0, rMaxSignal: arInputNormBounds[6], rMinSignal: arInputNormBounds[13], rNormTol: arInputNormTol[6], rMaxVal: arInputValBounds[6], rMinVal: arInputValBounds[13], tBoundErrorTime: T#5s, wWordSignal: awWordInputSignal[3], iIntSignal: emptyIntSignals[3], rMeasurement: arLinearizedInputSIgnals[3], xAssignmentFlag => axFaultFlags[1])
NETWORK 13
	fbflowassign:FB_AssignAnalog(EN: *, xWord: TRUE, wWordInput: dummywordsignals[4], iIntInput: 0, rMaxSignal: arInputNormBounds[7], rMinSignal: arInputNormBounds[14], rNormTol: arInputNormTol[7], rMaxVal: arInputValBounds[7], rMinVal: arInputValBounds[14], tBoundErrorTime: T#5s, wWordSignal: awWordInputSignal[4], iIntSignal: emptyIntSignals[4], rMeasurement: arLinearizedInputSIgnals[4], xAssignmentFlag => axFaultFlags[2])
NETWORK 14
	fbwaterlevellow:FB_AssignDigital(EN: *, xBoolSignal: dummyboolsignals[1], tDebounceTime: T#2S, xDetectRisingEdge: FALSE, xDetectFallingEdge: FALSE, xDebouncedSignal: axBoolDebouncedInputSignal[1], xOutputSignal => axBoolInputSignal[1])
NETWORK 15
	fbwaterlevellowlowlow:FB_AssignDigital(EN: *, xBoolSignal: dummyboolsignals[2], tDebounceTime: T#2S, xDetectRisingEdge: FALSE, xDetectFallingEdge: FALSE, xDebouncedSignal: axBoolDebouncedInputSignal[2], xOutputSignal => axBoolInputSignal[2])
NETWORK 16
	fbpressure:FB_AssignDigital(EN: *, xBoolSignal: dummyboolsignals[3], tDebounceTime: T#2S, xDetectRisingEdge: FALSE, xDetectFallingEdge: FALSE, xDebouncedSignal: axBoolDebouncedInputSignal[3], xOutputSignal => axBoolInputSignal[3])
NETWORK 17
	fbcondwarning:FB_AssignDigital(EN: *, xBoolSignal: dummyboolsignals[4], tDebounceTime: T#2S, xDetectRisingEdge: FALSE, xDetectFallingEdge: FALSE, xDebouncedSignal: axBoolDebouncedInputSignal[4], xOutputSignal => axBoolInputSignal[4])
NETWORK 18
	fbcondfault:FB_AssignDigital(EN: *, xBoolSignal: dummyboolsignals[5], tDebounceTime: T#2S, xDetectRisingEdge: FALSE, xDetectFallingEdge: FALSE, xDebouncedSignal: axBoolDebouncedInputSignal[5], xOutputSignal => axBoolInputSignal[5])
NETWORK 19
	fbpvv:FB_PumpValueValidation(EN: *, xPoorReadPrimary: axInputSignalFlags[1], xPoorReadSecondary: axInputSignalFlags[2], xPrimaryPumpActive: axActivePumps[1], xSecondaryPumpActive: axActivePumps[2], rPrimaryPower: arMultiSignals[1], rSecondaryPower: arMultiSignals[2], rPumpPower: arLinearizedInputSIgnals[1], xRequestPumpTurnover => axAutoTurnoverRequests[1])
NETWORK 20
	fbtsa:FB_TempSystemAlignment(EN: *, rTemp1: arMultiSignals[3], rTemp2: arMultiSignals[4], rTemp3: arMultiSignals[5], xRTD1Flag: axInputSignalFlags[3], xRTD2Flag: axInputSignalFlags[4], xRTD3Flag: axInputSignalFlags[5], rMeasuredTemp => arLinearizedInputSIgnals[2])
NETWORK 21
	fbcheckwaterlevel:FB_CheckWaterLevel(EN: *, xLow: axBoolDebouncedInputSignal[1], xLowLow: axBoolDebouncedInputSignal[2], xVesselLevelLow => axSystemAlerts[6], xVesselLevelCritical => axFaultFlags[4], xVesselLevelSensorFailure => axFaultFlags[5])
NETWORK 22
	fbcheckconductivity:FB_CheckConductivity(EN: *, xConductivityBadRead: axFaultFlags[1], xConductivityAlarmTrip: axBoolInputSignal[4], xConductivityFaultTrip: axBoolInputSignal[5], rConductivityMeasurement: arLinearizedInputSIgnals[3], rConductivityAlarmThreshold: 50, rConductivityFaultThreshold: 60, tHysteresisTime: T#100ms, tAlignmentTime: T#100ms, xConductivitySensorError => axFaultFlags[6], xConductivityWarning => axSystemAlerts[7], xConductivityAlert => axFaultFlags[7])
NETWORK 23
	fbpowerpressureflowthreshold:FB_PowerPressureFlowThreshold(EN: *, rPumpPowerLowThreshold: 30, rPumpPower: arLinearizedInputSignals[1], rFlow: arLinearizedInputSignals[4], rFlowLowThreshold: 30, xPressureLowInput: axBoolDebouncedInputSignal[3], tHysteresisTime: T#100ms, xPumpPowerLow => axSystemAlerts[8], xFlowLow => axSystemAlerts[9], xPressureLowFlag => axSystemAlerts[10])
NETWORK 24
	fbpowerpressureflowvote:FB_PowerPressureFlowVote(EN: *, xLowPressure: axSystemAlerts[10], xLowFlow: axSystemAlerts[9], xLowPower: axSystemAlerts[8], xPrimaryPumpActive: axActivePumps[1], xSecondaryPumpActive: axActivePumps[2], xSystemInitializing: axSystemAlerts[3], xSystemShuttingDown: axSystemAlerts[2], xSystemOn: axSystemAlerts[1], xPrimaryHydraulicFailure: axHydraulicFailures[1], xSecondaryHydraulicFailure: axHydraulicFailures[2], xRequestPumpSwitch => axAutoTurnoverRequests[2])
NETWORK 25
	fbtempboundcheck:FB_TemperatureBoundCheck(EN: *, rSystemTemperature: arLinearizedInputSignals[2], rTempFaultMin: 10, rTempFaultMax: 90, rTempAlarmMin: 30, rTempAlarmMax: 50, tWarningTime: T#100ms, tFailureTime: T#100ms, xAwaitInit: axSystemAlerts[3], xAwaitCalibration: axSystemAlerts[4], xSystemOn: axSystemAlerts[1], xSystemShuttingDown: axSystemAlerts[2], xTemperatureWarning: axSystemAlerts[11], xTemperatureFailure: axFaultFlags[8])
NETWORK 26
	fbmatl:FB_MasterAutoTurnoverLink(EN: *, xPrimaryAutoTurnover: axAutoTurnoverRequests[1], xSecondaryAutoTurnOver: axAutoTurnoverRequests[2], xMasterAutoTurnover => xMasterAutoTurnoverRequest)
NETWORK 27
	fbpsc:FB_PumpSwitchControl(EN: *, xSystemShutdownInProgress: axSystemAlerts[2], xSystemOn: axSystemAlerts[1], xSystemCali: axSystemAlerts[4], xSystemInit: axSystemAlerts[3], ManualSwitchRequest: USERTurnoverRequest, AutomaticSwitchRequest: xMasterAutoTurnoverRequest, SimplexMode: axSystemAlerts[5], InitiateSwitch: xMasterTurnoverRequest, DuplexFailure: axFaultFlags[3])
NETWORK 28
	fbsil:FB_SwitchInitLink(EN: *, xShutdownInProgress: axSystemAlerts[2], xSimplexMode: axSystemAlerts[5], xBeginSystemInitialization: USERMasterStart, xInitializePumpSwitch: xMasterTurnoverRequest, xSystemOn: axSystemAlerts[1])
_END_LD_
(* the same logic as Structured Text *)
(* Network 1 *)
fbsysstart(xEnable := TRUE, tInitilizationTime := T#3S, tCalibrationTime := T#3S, xSystemShutdownInProgress := axSystemAlerts[2], xBeginSystemInitialization := USERMasterStart, axInstrumentFlags := axFaultFlags, xSystemOn := axSystemAlerts[1], xFaultACK := USERAcknowledgeFault, xFaultExists := xMasterFault, xSystemInitializing := axSystemAlerts[3], xSystemCalibrating := axSystemAlerts[4]);
(* Network 2 *)
fbstop(xEnable := TRUE, xFaultExists := xMasterFault, tSDTime := T#2000MS, xSystemShutdownInProgress := axSystemAlerts[2], xSystemOn := axSystemAlerts[1], xSystemInitializing := axSystemAlerts[3], xSystemCalibrating := axSystemAlerts[4], xForceShutdown := USERShutdown);
(* Network 3 *)
fbfaultcheck(xEnable := TRUE, axInstrumentFlags := axFaultFlags, xFaultExists := xMasterFault);
(* Network 4 *)
fbpc(EN := TRUE, xSystemShutdownInProgress := axSystemAlerts[2], xSystemON := axSystemAlerts[1], xSystemInitializing := axSystemAlerts[3], xPrimaryPumpActive := axActivePumps[1], xSecondaryPumpActive := axActivePumps[2], xInitiatePumpSwitch := USERTurnoverRequest, xBeginSystemInitialization := USERMasterStart);
(* Network 5 *)
fbfc(EN := TRUE, xSystemShuttingDown := axSystemAlerts[2], xEnableFans := axSystemAlerts[16], xForceFan1On := axSystemAlerts[12], xForceFan2On := axSystemAlerts[13], xManualControl := axSystemAlerts[15]);
axActiveFans[1] := fbfc.xCoolantFan1;
axActiveFans[2] := fbfc.xCoolantFan2;
(* Network 6 *)
fbtcoo(EN := TRUE, rMeasuredTemp := arLinearizedInputSignals[2], rLowThreshold := 37, rHighThreshold := 42, xSystemInitializing := axSystemAlerts[3], xSystemShuttingDown := axSystemAlerts[2], xManualControl := axSystemAlerts[15], SystemOn := axSystemAlerts[1], xForceThroughput := axSystemAlerts[14]);
rPercentValveOpen := fbtcoo.rOutput;
axSystemAlerts[16] := fbtcoo.xEnableFans;
(* Network 7 *)
fbpump1assign(EN := TRUE, xWord := TRUE, wWordInput := dummywordsignals[1], iIntInput := 0, rMaxSignal := arInputNormBounds[1], rMinSignal := arInputNormBounds[8], rNormTol := arInputNormTol[1], rMaxVal := arInputValBounds[1], rMinVal := arInputValBounds[8], tBoundErrorTime := T#5s, wWordSignal := awWordInputSignal[1], iIntSignal := emptyIntSignals[1], rMeasurement := arMultiSignals[1]);
axInputSignalFlags[1] := fbpump1assign.xAssignmentFlag;
(* Network 8 *)
fbpump2assign(EN := TRUE, xWord := TRUE, wWordInput := dummywordsignals[2], iIntInput := 0, rMaxSignal := arInputNormBounds[2], rMinSignal := arInputNormBounds[9], rNormTol := arInputNormTol[2], rMaxVal := arInputValBounds[2], rMinVal := arInputValBounds[9], tBoundErrorTime := T#5s, wWordSignal := awWordInputSignal[2], iIntSignal := emptyIntSignals[2], rMeasurement := arMultiSignals[2]);
axInputSignalFlags[2] := fbpump2assign.xAssignmentFlag;
(* Network 9 *)
fbrtd1assign(EN := TRUE, xWord := FALSE, wWordInput := 0, iIntInput := dummyintsignals[1], rMaxSignal := arInputNormBounds[3], rMinSignal := arInputNormBounds[10], rNormTol := arInputNormTol[3], rMaxVal := arInputValBounds[3], rMinVal := arInputValBounds[10], tBoundErrorTime := T#5s, wWordSignal := emptyWordSignals[1], iIntSignal := aiIntInputSignal[1], rMeasurement := arMultiSignals[3]);
axInputSignalFlags[3] := fbrtd1assign.xAssignmentFlag;
(* Network 10 *)
fbrtd2assign(EN := TRUE, xWord := FALSE, wWordInput := 0, iIntInput := dummyintsignals[2], rMaxSignal := arInputNormBounds[4], rMinSignal := arInputNormBounds[11], rNormTol := arInputNormTol[4], rMaxVal := arInputValBounds[4], rMinVal := arInputValBounds[11], tBoundErrorTime := T#5s, wWordSignal := emptyWordSignals[2], iIntSignal := aiIntInputSignal[2], rMeasurement := arMultiSignals[4]);
axInputSignalFlags[4] := fbrtd2assign.xAssignmentFlag;
(* Network 11 *)
fbrtd3assign(EN := TRUE, xWord := FALSE, wWordInput := 0, iIntInput := dummyintsignals[3], rMaxSignal := arInputNormBounds[5], rMinSignal := arInputNormBounds[12], rNormTol := arInputNormTol[5], rMaxVal := arInputValBounds[5], rMinVal := arInputValBounds[12], tBoundErrorTime := T#5s, wWordSignal := emptyWordSignals[3], iIntSignal := aiIntInputSignal[3], rMeasurement := arMultiSignals[5]);
axInputSignalFlags[5] := fbrtd3assign.xAssignmentFlag;
(* Network 12 *)
fbcondassign(EN := TRUE, xWord := TRUE, wWordInput := dummywordsignals[3], iIntInput := 0, rMaxSignal := arInputNormBounds[6], rMinSignal := arInputNormBounds[13], rNormTol := arInputNormTol[6], rMaxVal := arInputValBounds[6], rMinVal := arInputValBounds[13], tBoundErrorTime := T#5s, wWordSignal := awWordInputSignal[3], iIntSignal := emptyIntSignals[3], rMeasurement := arLinearizedInputSIgnals[3]);
axFaultFlags[1] := fbcondassign.xAssignmentFlag;
(* Network 13 *)
fbflowassign(EN := TRUE, xWord := TRUE, wWordInput := dummywordsignals[4], iIntInput := 0, rMaxSignal := arInputNormBounds[7], rMinSignal := arInputNormBounds[14], rNormTol := arInputNormTol[7], rMaxVal := arInputValBounds[7], rMinVal := arInputValBounds[14], tBoundErrorTime := T#5s, wWordSignal := awWordInputSignal[4], iIntSignal := emptyIntSignals[4], rMeasurement := arLinearizedInputSIgnals[4]);
axFaultFlags[2] := fbflowassign.xAssignmentFlag;
(* Network 14 *)
fbwaterlevellow(EN := TRUE, xBoolSignal := dummyboolsignals[1], tDebounceTime := T#2S, xDetectRisingEdge := FALSE, xDetectFallingEdge := FALSE, xDebouncedSignal := axBoolDebouncedInputSignal[1]);
axBoolInputSignal[1] := fbwaterlevellow.xOutputSignal;
(* Network 15 *)
fbwaterlevellowlowlow(EN := TRUE, xBoolSignal := dummyboolsignals[2], tDebounceTime := T#2S, xDetectRisingEdge := FALSE, xDetectFallingEdge := FALSE, xDebouncedSignal := axBoolDebouncedInputSignal[2]);
axBoolInputSignal[2] := fbwaterlevellowlowlow.xOutputSignal;
(* Network 16 *)
fbpressure(EN := TRUE, xBoolSignal := dummyboolsignals[3], tDebounceTime := T#2S, xDetectRisingEdge := FALSE, xDetectFallingEdge := FALSE, xDebouncedSignal := axBoolDebouncedInputSignal[3]);
axBoolInputSignal[3] := fbpressure.xOutputSignal;
(* Network 17 *)
fbcondwarning(EN := TRUE, xBoolSignal := dummyboolsignals[4], tDebounceTime := T#2S, xDetectRisingEdge := FALSE, xDetectFallingEdge := FALSE, xDebouncedSignal := axBoolDebouncedInputSignal[4]);
axBoolInputSignal[4] := fbcondwarning.xOutputSignal;
(* Network 18 *)
fbcondfault(EN := TRUE, xBoolSignal := dummyboolsignals[5], tDebounceTime := T#2S, xDetectRisingEdge := FALSE, xDetectFallingEdge := FALSE, xDebouncedSignal := axBoolDebouncedInputSignal[5]);
axBoolInputSignal[5] := fbcondfault.xOutputSignal;
(* Network 19 *)
fbpvv(EN := TRUE, xPoorReadPrimary := axInputSignalFlags[1], xPoorReadSecondary := axInputSignalFlags[2], xPrimaryPumpActive := axActivePumps[1], xSecondaryPumpActive := axActivePumps[2], rPrimaryPower := arMultiSignals[1], rSecondaryPower := arMultiSignals[2], rPumpPower := arLinearizedInputSIgnals[1]);
axAutoTurnoverRequests[1] := fbpvv.xRequestPumpTurnover;
(* Network 20 *)
fbtsa(EN := TRUE, rTemp1 := arMultiSignals[3], rTemp2 := arMultiSignals[4], rTemp3 := arMultiSignals[5], xRTD1Flag := axInputSignalFlags[3], xRTD2Flag := axInputSignalFlags[4], xRTD3Flag := axInputSignalFlags[5]);
arLinearizedInputSIgnals[2] := fbtsa.rMeasuredTemp;
(* Network 21 *)
fbcheckwaterlevel(EN := TRUE, xLow := axBoolDebouncedInputSignal[1], xLowLow := axBoolDebouncedInputSignal[2]);
axSystemAlerts[6] := fbcheckwaterlevel.xVesselLevelLow;
axFaultFlags[4] := fbcheckwaterlevel.xVesselLevelCritical;
axFaultFlags[5] := fbcheckwaterlevel.xVesselLevelSensorFailure;
(* Network 22 *)
fbcheckconductivity(EN := TRUE, xConductivityBadRead := axFaultFlags[1], xConductivityAlarmTrip := axBoolInputSignal[4], xConductivityFaultTrip := axBoolInputSignal[5], rConductivityMeasurement := arLinearizedInputSIgnals[3], rConductivityAlarmThreshold := 50, rConductivityFaultThreshold := 60, tHysteresisTime := T#100ms, tAlignmentTime := T#100ms);
axFaultFlags[6] := fbcheckconductivity.xConductivitySensorError;
axSystemAlerts[7] := fbcheckconductivity.xConductivityWarning;
axFaultFlags[7] := fbcheckconductivity.xConductivityAlert;
(* Network 23 *)
fbpowerpressureflowthreshold(EN := TRUE, rPumpPowerLowThreshold := 30, rPumpPower := arLinearizedInputSignals[1], rFlow := arLinearizedInputSignals[4], rFlowLowThreshold := 30, xPressureLowInput := axBoolDebouncedInputSignal[3], tHysteresisTime := T#100ms);
axSystemAlerts[8] := fbpowerpressureflowthreshold.xPumpPowerLow;
axSystemAlerts[9] := fbpowerpressureflowthreshold.xFlowLow;
axSystemAlerts[10] := fbpowerpressureflowthreshold.xPressureLowFlag;
(* Network 24 *)
fbpowerpressureflowvote(EN := TRUE, xLowPressure := axSystemAlerts[10], xLowFlow := axSystemAlerts[9], xLowPower := axSystemAlerts[8], xPrimaryPumpActive := axActivePumps[1], xSecondaryPumpActive := axActivePumps[2], xSystemInitializing := axSystemAlerts[3], xSystemShuttingDown := axSystemAlerts[2], xSystemOn := axSystemAlerts[1], xPrimaryHydraulicFailure := axHydraulicFailures[1], xSecondaryHydraulicFailure := axHydraulicFailures[2]);
axAutoTurnoverRequests[2] := fbpowerpressureflowvote.xRequestPumpSwitch;
(* Network 25 *)
fbtempboundcheck(EN := TRUE, rSystemTemperature := arLinearizedInputSignals[2], rTempFaultMin := 10, rTempFaultMax := 90, rTempAlarmMin := 30, rTempAlarmMax := 50, tWarningTime := T#100ms, tFailureTime := T#100ms, xAwaitInit := axSystemAlerts[3], xAwaitCalibration := axSystemAlerts[4], xSystemOn := axSystemAlerts[1], xSystemShuttingDown := axSystemAlerts[2], xTemperatureWarning := axSystemAlerts[11], xTemperatureFailure := axFaultFlags[8]);
(* Network 26 *)
fbmatl(EN := TRUE, xPrimaryAutoTurnover := axAutoTurnoverRequests[1], xSecondaryAutoTurnOver := axAutoTurnoverRequests[2]);
xMasterAutoTurnoverRequest := fbmatl.xMasterAutoTurnover;
(* Network 27 *)
fbpsc(EN := TRUE, xSystemShutdownInProgress := axSystemAlerts[2], xSystemOn := axSystemAlerts[1], xSystemCali := axSystemAlerts[4], xSystemInit := axSystemAlerts[3], ManualSwitchRequest := USERTurnoverRequest, AutomaticSwitchRequest := xMasterAutoTurnoverRequest, SimplexMode := axSystemAlerts[5], InitiateSwitch := xMasterTurnoverRequest, DuplexFailure := axFaultFlags[3]);
(* Network 28 *)
fbsil(EN := TRUE, xShutdownInProgress := axSystemAlerts[2], xSimplexMode := axSystemAlerts[5], xBeginSystemInitialization := USERMasterStart, xInitializePumpSwitch := xMasterTurnoverRequest, xSystemOn := axSystemAlerts[1]);
END_PROGRAM

(* POU Instrument Control/Check Control/FB_CheckWaterLevel, ST *)
FUNCTION_BLOCK FB_CheckWaterLevel
VAR_INPUT
	EN: BOOL;
	xLow: BOOL;
	xLowLow: BOOL;
END_VAR
VAR_OUTPUT
	END: BOOL;
	xVesselLevelLow: BOOL;
	xVesselLevelCritical: BOOL;
	xVesselLevelSensorFailure: BOOL;
END_VAR
VAR
END_VAR
END := FALSE;
IF EN = FALSE THEN
	RETURN;
END_IF

IF xLow AND xLowLow = FALSE THEN
	xVesselLevelLow := TRUE;
	xVesselLevelCritical := FALSE;
	xVesselLevelSensorFailure := FALSE;
ELSIF xLow  AND xLowLow THEN
	xVesselLevelLow := TRUE;
	xVesselLevelCritical := TRUE;
	xVesselLevelSensorFailure := FALSE;
ELSIF xLowLow AND xLow <> TRUE THEN
	xVesselLevelLow := FALSE;
	xVesselLevelCritical := FALSE;
	xVesselLevelSensorFailure := TRUE;
ELSE
	xVesselLevelLow := FALSE;
	xVesselLevelCritical := FALSE;
	xVesselLevelSensorFailure := FALSE;
END_IF

END := TRUE;
END_FUNCTION_BLOCK

(* POU Instrument Control/Check Control/FB_CheckConductivity, ST *)
FUNCTION_BLOCK FB_CheckConductivity
VAR_INPUT
	EN: BOOL;
	xConductivityBadRead: BOOL;
	xConductivityAlarmTrip: BOOL;
	xConductivityFaultTrip: BOOL;
	rConductivityMeasurement: REAL;
	rConductivityAlarmThreshold: REAL;
	rConductivityFaultThreshold: REAL;
	tHysteresisTime: TIME;
	tAlignmentTime: TIME;
END_VAR
VAR_OUTPUT
	END: BOOL;
	xConductivitySensorError: BOOL;
	xConductivityWarning: BOOL;
	xConductivityAlert: BOOL;
END_VAR
VAR
	xConductivityAlarmBasedOnCalculations: BOOL;
	xConductivityFaultBasedOnCalculations: BOOL;
	iAlarmCount: INT;
	iFaultCount: INT;
	fbTON1: TON;
	fbTON2: TON;
	fbdebounce1: FB_DebounceSignal;
	fbdebounce2: FB_DebounceSignal;
	xConductivityMisalignmentErrorCandidate: BOOL;
END_VAR
END := FALSE;
IF EN = FALSE THEN
	RETURN;
END_IF

IF xConductivityBadRead THEN
	RETURN;
ELSE
	xConductivityAlarmBasedOnCalculations := F_BoundCheck(rInput := rConductivityMeasurement,
																	   xMaxCheck := TRUE,
																	   xMinCheck := FALSE,
																	   rMaxVariable :=  rConductivityAlarmThreshold,
																	   rMinVariable := 0,
																	   rTolerance := 0);
	fbdebounce1(EN := TRUE, xInput := xConductivityAlarmBasedOnCalculations, tDebounceTime := tHysteresisTime);

	xConductivityFaultBasedOnCalculations := F_BoundCheck(rInput := rConductivityMeasurement,
																	   xMaxCheck := TRUE,
																	   xMinCheck := FALSE,
																	   rMaxVariable :=  rConductivityFaultThreshold,
																	   rMinVariable := 0,
																	   rTolerance := 0);
	fbdebounce2(EN := TRUE, xInput := xConductivityFaultBasedOnCalculations, tDebounceTime := tHysteresisTime);

	iAlarmCount := BOOL_TO_INT(fbdebounce1.xOutput) + BOOL_TO_INT(xConductivityAlarmTrip);
	iFaultCount := BOOL_TO_INT(fbdebounce2.xOutput) + BOOL_TO_INT(xConductivityFaultTrip);

	IF iAlarmCount = 1 OR iFaultCount = 1 THEN
		xConductivityMisalignmentErrorCandidate := TRUE;
	END_IF
	IF (iFaultCount = 2 AND iAlarmCount = 1) THEN (*This guarantees that the sensor is not working*)
		xConductivitySensorError := TRUE;
	END_IF
	IF (iFaultCount = 2 AND iAlarmCount = 2) OR (iAlarmCount = 2) OR (iFaultCount = 0 AND iAlarmCount = 0) THEN
		xConductivityMisalignmentErrorCandidate := FALSE;
		xConductivitySensorError := FALSE;
	END_IF
	IF iAlarmCount = 2 THEN
		xConductivityWarning := TRUE;
	ELSIF iAlarmCount= 0 THEN
		xConductivityWarning := FALSE;
	END_IF
	IF iFaultCount = 2 THEN
		xConductivityAlert := TRUE;
	ELSIF iFaultCount = 0 THEN
		xConductivityAlert := FALSE;
	END_IF
END_IF
fbTON1(IN := xConductivityMisalignmentErrorCandidate, PT := tAlignmentTime);

IF fbTON1.Q THEN
	xConductivitySensorError := TRUE;
ELSE
	xConductivitySensorError := FALSE;
END_IF
END := TRUE;
END_FUNCTION_BLOCK

(* POU Functions/FB_DebounceSignal, ST *)
FUNCTION_BLOCK FB_DebounceSignal
VAR_INPUT
	EN: BOOL;
	xInput: BOOL;
	tDebounceTime: TIME;
END_VAR
VAR_OUTPUT
	END: BOOL;
	xOutput: BOOL;
END_VAR
VAR
	fbDebounceTimerON: TON;
	fbDebounceTimerOFF: TOF;
END_VAR
IF EN  = FALSE THEN
	RETURN;
END_IF

fbDebounceTimerON(IN := xInput, PT := tDebounceTime); (*Won't go to true until 50 ms of stability. Every false resets this timer*)

fbDebounceTimerOFF(IN := fbDebounceTimerON.Q, PT := tDebounceTime); (*Won't go to false until 50ms of stability. Every true resets this timer*)
xOutput  := fbDebounceTimerOFF.Q;

END := TRUE;
END_FUNCTION_BLOCK

(* POU Instrument Checking Functions/F_BoundCheck, ST *)
FUNCTION F_BoundCheck : BOOL
VAR_INPUT
	rInput: REAL;
	xMaxCheck: BOOL;
	xMinCheck: BOOL;
	rMaxVariable: REAL;
	rMinVariable: REAL;
	rTolerance: REAL;
END_VAR
VAR
	xPastBoundFlag: BOOL;
END_VAR
xPastBoundFlag := FALSE;
IF xMaxCheck = TRUE AND xMinCheck = TRUE THEN
	IF rInput > (rMaxVariable + rTolerance) THEN
		xPastBoundFlag := TRUE;
	ELSIF rInput < (rMinVariable - rTolerance) THEN
		xPastBoundFlag := TRUE;
	END_IF
ELSIF xMaxCheck = TRUE THEN
	IF rInput > (rMaxVariable + rTolerance) THEN
		xPastBoundFlag := TRUE;
	END_IF
ELSIF xMinCheck = TRUE THEN
	IF rInput < (rMinVariable - rTolerance) THEN
		xPastBoundFlag := TRUE;
	END_IF
END_IF

F_BoundCheck := xPastBoundFlag;
END_FUNCTION

(* POU Instrument Control/Check Control/FB_PowerPressureFlowThreshold, ST *)
FUNCTION_BLOCK FB_PowerPressureFlowThreshold
VAR_INPUT
	EN: BOOL;
	rPumpPowerLowThreshold: REAL;
	rPumpPower: REAL;
	rFlow: REAL;
	rFlowLowThreshold: REAL;
	xPressureLowInput: BOOL;
	tHysteresisTime: TIME;
END_VAR
VAR_OUTPUT
	END: BOOL;
	xPumpPowerLow: BOOL;
	xFlowLow: BOOL;
	xPressureLowFlag: BOOL;
END_VAR
VAR
	fbInitializeTimer: TON;
	xPumpPowerLowUF: BOOL;
	fbTON1: TON;
	xFlowLowUF: BOOL;
	fbTON2: TON;
	fbdebounce1: FB_DebounceSignal;
	fbdebounce2: FB_DebounceSignal;
END_VAR
IF EN = FALSE THEN
	RETURN;
END_IF
END := FALSE;
xPumpPowerLowUF := F_BoundCheck(rInput := rPumpPower,
										 xMaxCheck := FALSE,
										 xMinCheck := TRUE,
										 rMaxVariable :=  0,
										 rMinVariable := rPumpPowerLowThreshold,
										 rTolerance := 0);
fbdebounce1(EN := TRUE, xInput := xPumpPowerLowUF, tDebounceTime := tHysteresisTime);
xPumpPowerLow := fbdebounce1.xOutput;

xFlowLowUF := F_BoundCheck(rInput := rFlow,
										 xMaxCheck := FALSE,
										 xMinCheck := TRUE,
										 rMaxVariable :=  0,
										 rMinVariable := rFlowLowThreshold,
										 rTolerance := 0);
fbdebounce2(EN := TRUE, xInput := xFlowLowUF, tDebounceTime := tHysteresisTime);
xFlowLow := fbdebounce2.xOutput;


xPressureLowFlag := xPressureLowInput;

END := TRUE;
END_FUNCTION_BLOCK

(* POU Instrument Control/Check Control/FB_PowerPressureFlowVote, ST *)
FUNCTION_BLOCK FB_PowerPressureFlowVote
VAR_INPUT
	EN: BOOL;
	xLowPressure: BOOL;
	xLowFlow: BOOL;
	xLowPower: BOOL;
	xPrimaryPumpActive: BOOL;
	xSecondaryPumpActive: BOOL;
	xSystemInitializing: BOOL;
	xSystemShuttingDown: BOOL;
	xSystemOn: BOOL;
END_VAR
VAR_OUTPUT
	END: BOOL;
	xRequestPumpSwitch: BOOL;
END_VAR
VAR
	iBadCount: INT;
END_VAR
VAR_IN_OUT
	xPrimaryHydraulicFailure: BOOL;
	xSecondaryHydraulicFailure: BOOL;
END_VAR
IF EN = FALSE THEN
	RETURN;
END_IF
END := FALSE;
iBadCount := BOOL_TO_INT(xLowPressure) + BOOL_TO_INT(xLowFlow) + BOOL_TO_INT(xLowPower);

IF xSystemInitializing OR xSystemShuttingDown OR xSystemOn = FALSE THEN
	xRequestPumpSwitch := FALSE;
	END := TRUE;
	RETURN;
ELSE
	IF  (iBadCount > 1) THEN
		xRequestPumpSwitch := TRUE;
		IF (xPrimaryPumpActive = TRUE)  THEN
			xPrimaryHydraulicFailure := TRUE;
		ELSIF(xSecondaryPumpActive = TRUE) THEN
			xSecondaryHydraulicFailure := TRUE;
		END_IF
	ELSE
		xRequestPumpSwitch := FALSE;
	END_IF

END_IF
END := TRUE;
END_FUNCTION_BLOCK

(* POU Instrument Control/Check Control/FB_TemperatureBoundCheck, ST *)
FUNCTION_BLOCK FB_TemperatureBoundCheck
VAR_INPUT
	EN: BOOL;
	rSystemTemperature: REAL;
	rTempFaultMin: REAL;
	rTempFaultMax: REAL;
	rTempAlarmMin: REAL;
	rTempAlarmMax: REAL;
	tWarningTime: TIME;
	tFailureTime: TIME;
	xAwaitInit: BOOL;
	xAwaitCalibration: BOOL;
	xSystemOn: BOOL;
	xSystemShuttingDown: BOOL;
END_VAR
VAR_OUTPUT
	END: BOOL;
END_VAR
VAR
	xTempAlarm: BOOL;
	xTempFault: BOOL;
	fbTON1: TON;
	fbTON2: TON;
END_VAR
VAR_IN_OUT
	xTemperatureWarning: BOOL;
	xTemperatureFailure: BOOL;
END_VAR
END := FALSE;
IF EN = FALSE THEN
	RETURN;
END_IF
IF xAwaitInit OR xAwaitCalibration THEN
	xTempAlarm := FALSE;
	xTempFault := FALSE;
ELSIF xSystemShuttingDown OR xSystemOn = FALSE  THEN
	END := TRUE;
	RETURN;
ELSE
	xTempAlarm := F_BoundCheck(rInput := rSystemTemperature,
										 	xMaxCheck := TRUE,
										 	xMinCheck := TRUE,
										 	rMaxVariable := rTempAlarmMax,
										 	rMinVariable := rTempAlarmMin,
										 	rTolerance := 0);
	xTempFault := F_BoundCheck(rInput := rSystemTemperature,
										 	xMaxCheck := TRUE,
										 	xMinCheck := TRUE,
										 	rMaxVariable :=  rTempFaultMax,
										 	rMinVariable := rTempFaultMin,
										 	rTolerance := 0);
END_IF
fbTON1(IN := xTempAlarm, PT := tWarningTime);
fbTON2(IN := xTempFault, PT := tFailureTime);
xTemperatureWarning := fbTON1.Q;
xTemperatureFailure := fbTON2.Q;
END := TRUE;
END_FUNCTION_BLOCK

(* POU System Startup/FB_SystemStart, ST *)
FUNCTION_BLOCK FB_SystemStart
VAR_INPUT
	xEnable: BOOL;

	tInitilizationTime: TIME;
	tCalibrationTime: TIME;
	xSystemShutdownInProgress: BOOL;
END_VAR
VAR_OUTPUT
	xDone: BOOL;

END_VAR
VAR
	i: INT;

	fbInit: TON;
	fbCali: TON;
END_VAR
VAR_IN_OUT
	xBeginSystemInitialization: BOOL;
	axInstrumentFlags: ARRAY [1..25] OF BOOL;
	xSystemOn: BOOL;
	xFaultACK: BOOL;
	xFaultExists: BOOL;
	xSystemInitializing: BOOL;
	xSystemCalibrating: BOOL;
END_VAR
xDone := FALSE;
IF xEnable = FALSE THEN
	RETURN;
END_IF;

fbInit(IN := xSystemOn, PT := tInitilizationTime);
fbCali(IN:= fbInit.Q, PT := tCalibrationTime);

IF (xSystemShutdownInProgress = TRUE) OR (xBeginSystemInitialization = TRUE AND xFaultExists = TRUE AND xFaultAck = FALSE) OR (xBeginSystemInitialization = TRUE AND xFaultExists = FALSE AND xFaultAck = TRUE)  THEN
	xBeginSystemInitialization := FALSE;
	xDone  := TRUE;
	RETURN;
ELSIF (xBeginSystemInitialization = TRUE AND xFaultExists = TRUE AND xFaultACK = TRUE) THEN
	FOR i := 1 TO 25 DO
		axInstrumentFlags[i] := FALSE;
	END_FOR;
	xSystemOn := TRUE;
	xSystemInitializing := TRUE;
	xSystemCalibrating := TRUE;
	xFaultExists := FALSE;
	xFaultACK := FALSE;
ELSIF xBeginSystemInitialization = TRUE AND xFaultExists = FALSE AND xFaultACK = FALSE THEN
	xSystemOn := TRUE;
	xSystemInitializing := TRUE;
	xSystemCalibrating := TRUE;
END_IF

IF fbInit.Q = TRUE THEN
	xSystemInitializing := FALSE;
END_IF
IF fbCali.Q = TRUE THEN
	xSystemCalibrating := FALSE;
END_IF

xDone := TRUE;
END_FUNCTION_BLOCK

(* POU System Startup/FB_FaultCheck, ST *)
FUNCTION_BLOCK FB_FaultCheck
VAR_INPUT
	xEnable: BOOL;
	axInstrumentFlags: ARRAY [1..25] OF BOOL;
END_VAR
VAR_OUTPUT
	xDone: BOOL;

END_VAR
VAR
	i: INT;
END_VAR
VAR_IN_OUT
	xFaultExists: BOOL;
END_VAR
xDone := FALSE;
IF xEnable = FALSE THEN
	RETURN;
END_IF;
FOR i := 1 TO 15 DO
		IF axInstrumentFlags[i] = TRUE THEN
			xFaultExists := TRUE;
		END_IF;
END_FOR;
xDone := TRUE;
END_FUNCTION_BLOCK

(* POU System Startup/FB_SystemStop, ST *)
FUNCTION_BLOCK FB_SystemStop
VAR_INPUT
	xEnable: BOOL;

	xFaultExists: BOOL;
	tSDTime: TIME;
END_VAR
VAR_OUTPUT
	xDone: BOOL;

END_VAR
VAR
	xOFF: BOOL;
	fbSD: TON;

END_VAR

VAR_IN_OUT
	xSystemShutdownInProgress: BOOL;
	xSystemOn: BOOL;
	xSystemInitializing: BOOL;
	xSystemCalibrating: BOOL;
	xForceShutdown: BOOL;
END_VAR
xDone := FALSE;
IF xEnable = FALSE THEN
	xDone := TRUE;
	RETURN;
END_IF
fbSD(IN := 	xSystemShutdownInProgress, PT := tSDTime);
IF (xForceShutdown = FALSE AND xFaultExists = FALSE AND xSystemShutdownInProgress = FALSE AND xSystemOn = TRUE) OR xSystemOn = FALSE THEN
	RETURN;
ELSIF (xForceShutdown = TRUE OR xFaultExists = TRUE) AND (xSystemShutdownInProgress = FALSE) THEN
	xForceShutdown := FALSE;
	xSystemShutdownInProgress := TRUE;
	xSystemInitializing := FALSE;
	xSystemCalibrating := FALSE;
END_IF



IF fbSD.Q THEN
	xSystemShutdownInProgress := FALSE;
	xSystemOn := FALSE;
END_IF
xDone := TRUE;
END_FUNCTION_BLOCK

(* POU Instrument Control/FB_PumpSwitchControl, ST *)
FUNCTION_BLOCK FB_PumpSwitchControl
VAR_INPUT
	EN: BOOL;
	xSystemShutdownInProgress: BOOL;
	xSystemOn: BOOL;
	xSystemCali: BOOL;
	xSystemInit: BOOL;
END_VAR
VAR_OUTPUT
	END: BOOL;
END_VAR
VAR
END_VAR
VAR_IN_OUT
	ManualSwitchRequest: BOOL; {*Request Flags*}
	AutomaticSwitchRequest: BOOL; {*Request Flags*}
	SimplexMode: BOOL; {*SINCON Flag*}
	InitiateSwitch: BOOL;
	DuplexFailure: BOOL; {*Fault Flag*}
END_VAR
END := FALSE;
IF EN = FALSE THEN
	RETURN;
END_IF

IF ManualSwitchRequest = FALSE AND AutomaticSwitchRequest = FALSE THEN
	InitiateSwitch := FALSE;
	END := TRUE;
	RETURN;
ELSIF (ManualSwitchRequest = TRUE OR AutomaticSwitchRequest = TRUE) AND (xSystemShutdownInProgress OR xSystemOn = FALSE) THEN
	ManualSwitchRequest := FALSE;
	AutomaticSwitchRequest := FALSE;
	InitiateSwitch := FALSE;
ELSIF (AutomaticSwitchRequest = TRUE) AND (xSystemCali OR xSystemInit) THEN
	ManualSwitchRequest := FALSE;
	AutomaticSwitchRequest := FALSE;
	InitiateSwitch := FALSE;
ELSIF (AutomaticSwitchRequest = TRUE AND SimplexMode = FALSE)  THEN {*Autoswitch means something is wrong*}
	InitiateSwitch := TRUE;
	SimplexMode := TRUE;
	AutomaticSwitchRequest := FALSE;
ELSIF(ManualSwitchRequest = TRUE AND SimplexMode = FALSE) THEN
	InitiateSwitch := TRUE;
	ManualSwitchRequest := FALSE;
ELSIF (AutomaticSwitchRequest = TRUE AND SimplexMode = TRUE)  THEN {*Autoswitch means something is wrong*}
	DuplexFailure := TRUE; {*No pump to swtich back to*}
	AutomaticSwitchRequest := FALSE;
	InitiateSwitch := FALSE;
ELSIF (ManualSwitchRequest = TRUE AND SimplexMode = TRUE)  THEN {*Autoswitch means something is wrong*}
	 {*No pump to swtich back to*}
	ManualSwitchRequest := FALSE;
	InitiateSwitch := FALSE;
END_IF
ManualSwitchRequest := FALSE;
AutomaticSwitchRequest := FALSE;
END := TRUE;
END_FUNCTION_BLOCK

(* POU Instrument Control/FB_PumpControl, ST *)
FUNCTION_BLOCK FB_PumpControl
VAR_INPUT
	EN: BOOL;
	xSystemShutdownInProgress: BOOL;
	xSystemON: BOOL;
	xSystemInitializing: BOOL;
END_VAR
VAR_OUTPUT
	END: BOOL;

END_VAR
VAR
END_VAR
VAR_IN_OUT
	xPrimaryPumpActive: BOOL;
	xSecondaryPumpActive: BOOL;
	xInitiatePumpSwitch: BOOL;
	xBeginSystemInitialization: BOOL;
END_VAR
END := FALSE;
IF EN = FALSE THEN
	RETURN;
END_IF
IF (xSystemShutdownInProgress = TRUE OR xSystemON = FALSE) THEN
	xPrimaryPumpActive := FALSE;
	xSecondaryPumpActive := FALSE;
ELSIF xSystemInitializing = TRUE AND xBeginSystemInitialization = TRUE AND xPrimaryPumpActive = FALSE THEN
	xPrimaryPumpActive := TRUE;
	xSecondaryPumpActive := FALSE;
	xBeginSystemInitialization := FALSE;
ELSIF xSystemInitializing = TRUE AND xBeginSystemInitialization = TRUE AND xPrimaryPumpActive = TRUE THEN
	xPrimaryPumpActive := FALSE;
	xSecondaryPumpActive := TRUE;
	xBeginSystemInitialization := FALSE;
END_IF
END := TRUE;
END_FUNCTION_BLOCK

(* POU Instrument Control/FB_SwitchInitLink, ST *)
FUNCTION_BLOCK FB_SwitchInitLink
VAR_INPUT
	EN: BOOL;
	xShutdownInProgress: BOOL;
	xSimplexMode: BOOL;

END_VAR
VAR_OUTPUT
	END: BOOL;
END_VAR
VAR
END_VAR
VAR_IN_OUT
	xBeginSystemInitialization: BOOL;
	xInitializePumpSwitch: BOOL;
	xSystemOn: BOOL;
END_VAR
END := FALSE;
IF EN = FALSE THEN
	RETURN;
END_IF
IF xInitializePumpSwitch AND xShutdownInProgress = FALSE AND xSystemOn = TRUE THEN
	xInitializePumpSwitch := FALSE;
	xBeginSystemInitialization := TRUE;
	xSystemOn := FALSE;
ELSE
	xInitializePumpSwitch := FALSE;
	xBeginSystemInitialization := FALSE;
END_IF
END := TRUE;
END_FUNCTION_BLOCK

(* POU Data Conversion/Signal->Instrument/FB_AssignAnalog, LD *)
FUNCTION_BLOCK FB_AssignAnalog
VAR_INPUT
	EN: BOOL;
	xWord: BOOL;
	wWordInput: WORD;
	iIntInput: INT;
	rMaxSignal: REAL;
	rMinSignal: REAL;
	rNormTol: REAL;
	rMaxVal: REAL;
	rMinVal: REAL;
	tBoundErrorTime: TIME;
END_VAR
VAR_OUTPUT
	END: BOOL;
	xAssignmentFlag: BOOL;

END_VAR
VAR
	rSignal: REAL;
	rNormalizedSignal: REAL;
		rSignal1: REAL;
		rSignal2: REAL;
		rLastRead: REAL;
		rLinearizedSignal: REAL;
		xBoundError: BOOL;
		fbTON: TON;
		fbvalcap: FB_ValueCap;
	fbdebounce: FB_DebounceSignal;
END_VAR

VAR_IN_OUT
	wWordSignal: WORD;
	iIntSignal: INT;
	rMeasurement: REAL;
END_VAR
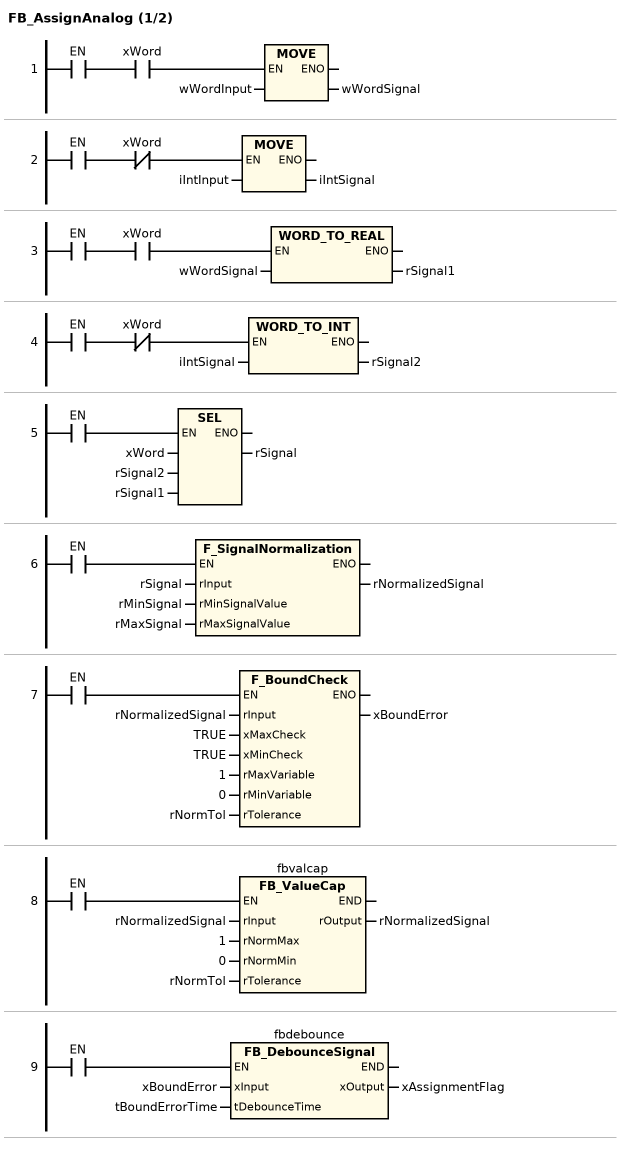
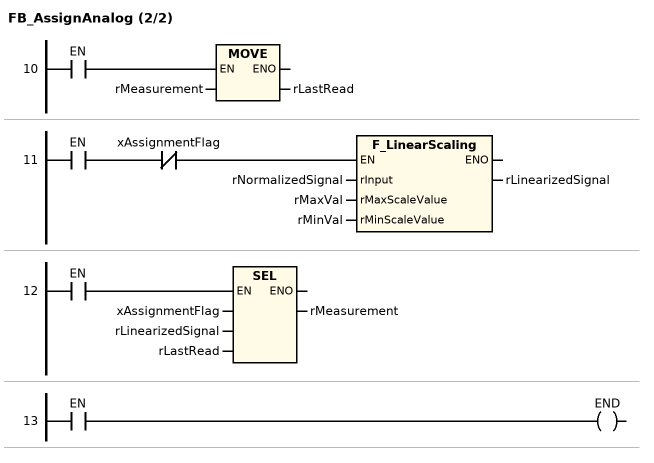
_LD_ (* Ladder Diagram *)
NETWORK 1
	[EN] - [xWord]
		EN --- MOVE(wWordInput) => wWordSignal
NETWORK 2
	[EN] - [/xWord]
		EN --- MOVE(iIntInput) => iIntSignal
NETWORK 3
	[EN] - [xWord]
		EN --- WORD_TO_REAL(wWordSignal) => rSignal1
NETWORK 4
	[EN] - [/xWord]
		EN --- WORD_TO_INT(iIntSignal) => rSignal2
NETWORK 5
	[EN]
		EN --- SEL(xWord, rSignal2, rSignal1) => rSignal
NETWORK 6
	[EN]
		EN --- F_SignalNormalization(rInput: rSignal, rMinSignalValue: rMinSignal, rMaxSignalValue: rMaxSignal) => rNormalizedSignal
NETWORK 7
	[EN]
		EN --- F_BoundCheck(rInput: rNormalizedSignal, xMaxCheck: TRUE, xMinCheck: TRUE, rMaxVariable: 1, rMinVariable: 0, rTolerance: rNormTol) => xBoundError
NETWORK 8
	[EN] - fbvalcap:FB_ValueCap(EN: *, rInput: rNormalizedSignal, rNormMax: 1, rNormMin: 0, rTolerance: rNormTol, rOutput => rNormalizedSignal)
NETWORK 9
	[EN] - fbdebounce:FB_DebounceSignal(EN: *, xInput: xBoundError, tDebounceTime: tBoundErrorTime, xOutput => xAssignmentFlag)
NETWORK 10
	[EN]
		EN --- MOVE(rMeasurement) => rLastRead
NETWORK 11
	[EN] - [/xAssignmentFlag]
		EN --- F_LinearScaling(rInput: rNormalizedSignal, rMaxScaleValue: rMaxVal, rMinScaleValue: rMinVal) => rLinearizedSignal
NETWORK 12
	[EN]
		EN --- SEL(xAssignmentFlag, rLinearizedSignal, rLastRead) => rMeasurement
NETWORK 13
	[EN] --- (END)
_END_LD_
(* the same logic as Structured Text *)
(* Network 1 *)
IF EN AND xWord THEN
	wWordSignal := wWordInput;
END_IF;
(* Network 2 *)
IF EN AND NOT xWord THEN
	iIntSignal := iIntInput;
END_IF;
(* Network 3 *)
IF EN AND xWord THEN
	rSignal1 := WORD_TO_REAL(wWordSignal);
END_IF;
(* Network 4 *)
IF EN AND NOT xWord THEN
	rSignal2 := WORD_TO_INT(iIntSignal);
END_IF;
(* Network 5 *)
IF EN THEN
	rSignal := SEL(xWord, rSignal2, rSignal1);
END_IF;
(* Network 6 *)
IF EN THEN
	rNormalizedSignal := F_SignalNormalization(rInput := rSignal, rMinSignalValue := rMinSignal, rMaxSignalValue := rMaxSignal);
END_IF;
(* Network 7 *)
IF EN THEN
	xBoundError := F_BoundCheck(rInput := rNormalizedSignal, xMaxCheck := TRUE, xMinCheck := TRUE, rMaxVariable := 1, rMinVariable := 0, rTolerance := rNormTol);
END_IF;
(* Network 8: see the listing above *)
(* Network 9: see the listing above *)
(* Network 10 *)
IF EN THEN
	rLastRead := rMeasurement;
END_IF;
(* Network 11 *)
IF EN AND NOT xAssignmentFlag THEN
	rLinearizedSignal := F_LinearScaling(rInput := rNormalizedSignal, rMaxScaleValue := rMaxVal, rMinScaleValue := rMinVal);
END_IF;
(* Network 12 *)
IF EN THEN
	rMeasurement := SEL(xAssignmentFlag, rLinearizedSignal, rLastRead);
END_IF;
(* Network 13 *)
END := EN;
END_FUNCTION_BLOCK

(* POU Functions/FB_ValueCap, ST *)
FUNCTION_BLOCK FB_ValueCap
VAR_INPUT
	EN: BOOL;
	rInput: REAL;
	rNormMax: REAL;
	rNormMin: REAL;
	rTolerance: REAL;
END_VAR
VAR_OUTPUT
	END: BOOL;
	rOutput: REAL;
END_VAR
VAR
	rLastRead: REAL := 0;
END_VAR
IF (rInput > rNormMax + rTolerance) OR (rInput < rNormMin - rTolerance) THEN
	rOutput  := rLastRead;
ELSIF (rInput > 1) THEN
	rOutput := 1;
	rLastRead := 1;
ELSIF (rInput < 0) THEN
	rOutput := 0;
	rLastRead := 0;
ELSE
	rOutput := rInput;
	rLastRead := rInput;
END_IF
END_FUNCTION_BLOCK

(* POU Functions/F_SignalNormalization, ST *)
FUNCTION F_SignalNormalization : REAL
VAR_INPUT
	rInput: REAL;
	rMinSignalValue: REAL;
	rMaxSignalValue: REAL;
END_VAR
VAR
END_VAR
IF rMinSignalValue > rMaxSignalValue OR rMinSignalValue = rMaxSignalValue THEN
	F_SignalNormalization := 0;
ELSE
	F_SignalNormalization  := ((rInput - rMinSignalValue)) / (rMaxSignalValue - rMinSignalValue);
END_IF
;
END_FUNCTION

(* POU Functions/F_LinearScaling, ST *)
FUNCTION F_LinearScaling : REAL
VAR_INPUT
	rInput: REAL;
	rMaxScaleValue: REAL;
	rMinScaleValue: REAL;
END_VAR
VAR
END_VAR
IF rMaxScaleValue <  rMinScaleValue OR rMaxScaleValue = rMinScaleValue THEN
	F_LinearScaling := 0;
ELSE
	F_LinearScaling := rInput * (rMaxScaleValue - rMinScaleValue) + rMinScaleValue;
END_IF
END_FUNCTION

(* POU Data Conversion/Signal->Instrument/FB_AssignDigital, LD *)
FUNCTION_BLOCK FB_AssignDigital
VAR_INPUT
	EN: BOOL;
	xBoolSignal: BOOL;
	tDebounceTime: TIME;
	xDetectRisingEdge: BOOL;
	xDetectFallingEdge: BOOL;
END_VAR
VAR_OUTPUT
	DONE: BOOL;
	xOutputSignal: BOOL;

END_VAR
VAR

	fbRise: R_TRIG;
	fbRTrig: R_TRIG;
	xSignalRise: BOOL;
	fbFTrig: F_TRIG;
	xSignalFall: BOOL;
	xEdgeSignal1: BOOL;
	xEdgeSignal: BOOL;
	fbdesig: FB_DebounceSignal;

END_VAR
VAR_IN_OUT
	xDebouncedSignal: BOOL;
END_VAR
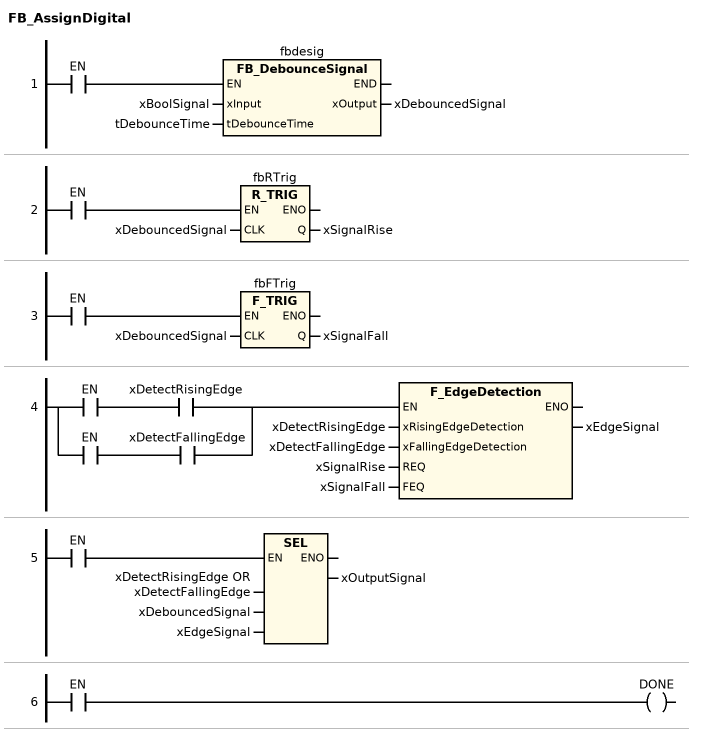
_LD_ (* Ladder Diagram *)
NETWORK 1
	[EN] - fbdesig:FB_DebounceSignal(EN: *, xInput: xBoolSignal, tDebounceTime: tDebounceTime, xOutput => xDebouncedSignal)
NETWORK 2
	[EN]
		EN --- fbRTrig:R_TRIG(CLK: xDebouncedSignal) => xSignalRise
NETWORK 3
	[EN]
		EN --- fbFTrig:F_TRIG(CLK: xDebouncedSignal) => xSignalFall
NETWORK 4
	{ [EN] - [xDetectRisingEdge] | [EN] - [xDetectFallingEdge] }
		EN --- F_EdgeDetection(xRisingEdgeDetection: xDetectRisingEdge, xFallingEdgeDetection: xDetectFallingEdge, REQ: xSignalRise, FEQ: xSignalFall) => xEdgeSignal
NETWORK 5
	[EN]
		EN --- SEL(xDetectRisingEdge OR xDetectFallingEdge, xDebouncedSignal, xEdgeSignal) => xOutputSignal
NETWORK 6
	[EN] --- (DONE)
_END_LD_
(* the same logic as Structured Text *)
(* Network 1: see the listing above *)
(* Network 2 *)
IF EN THEN
	fbRTrig(CLK := xDebouncedSignal);
	xSignalRise := fbRTrig.Q;
END_IF;
(* Network 3 *)
IF EN THEN
	fbFTrig(CLK := xDebouncedSignal);
	xSignalFall := fbFTrig.Q;
END_IF;
(* Network 4 *)
IF EN AND xDetectRisingEdge OR EN AND xDetectFallingEdge THEN
	xEdgeSignal := F_EdgeDetection(xRisingEdgeDetection := xDetectRisingEdge, xFallingEdgeDetection := xDetectFallingEdge, REQ := xSignalRise, FEQ := xSignalFall);
END_IF;
(* Network 5 *)
IF EN THEN
	xOutputSignal := SEL(xDetectRisingEdge OR xDetectFallingEdge, xDebouncedSignal, xEdgeSignal);
END_IF;
(* Network 6 *)
DONE := EN;
END_FUNCTION_BLOCK

(* POU Functions/F_EdgeDetection, ST *)
FUNCTION F_EdgeDetection : BOOL
VAR_INPUT
	xRisingEdgeDetection: BOOL;
	xFallingEdgeDetection: BOOL;
	REQ: BOOL;
	FEQ: BOOL;
END_VAR
VAR
END_VAR
IF xRisingEdgeDetection = TRUE AND xFallingEdgeDetection = TRUE THEN
	F_EdgeDetection := REQ OR FEQ; (*Are we detecing if this goes from False to True. When we detect this, caputre it*)
ELSIF xFallingEdgeDetection = TRUE THEN
	F_EdgeDetection := FEQ; (*Same as above but Vice Versa. Note that you can have both!*)
ELSIF xRisingEdgeDetection = TRUE THEN
	F_EdgeDetection  := REQ;
END_IF
END_FUNCTION

(* POU FB_PumpValueValidation, ST *)
FUNCTION_BLOCK FB_PumpValueValidation
VAR_INPUT
	EN: BOOL;
	xPoorReadPrimary: BOOL;
	xPoorReadSecondary: BOOL;
	xPrimaryPumpActive: BOOL;
	xSecondaryPumpActive: BOOL;
	rPrimaryPower: REAL;
	rSecondaryPower: REAL;
END_VAR
VAR_OUTPUT
	END: BOOL;
	xRequestPumpTurnover: BOOL;
END_VAR
VAR
	rLastPower: REAL;
END_VAR
VAR_IN_OUT
	rPumpPower: REAL;

END_VAR
END := FALSE;
IF EN = FALSE THEN
	RETURN;
END_IF

IF (xPoorReadPrimary AND xPrimaryPumpActive) OR (xPoorReadSecondary AND xSecondaryPumpActive) THEN
	xRequestPumpTurnover := TRUE;
	rPumpPower := rLastPower;
ELSE
	xRequestPumpTurnover := FALSE;
	IF xPrimaryPumpActive THEN
		rLastPower := rPumpPower;
		rPumpPower := rPrimaryPower;
	ELSIF xSecondaryPumpActive THEN
		rLastPower := rPumpPower;
		rPumpPower := rSecondaryPower;
	END_IF
END_IF
END := TRUE;
END_FUNCTION_BLOCK

(* POU Data Conversion/Instrument->System/FB_TempSystemAlignment, ST *)
FUNCTION_BLOCK FB_TempSystemAlignment
VAR_INPUT
	EN: BOOL;
	rTemp1: REAL;
	rTemp2: REAL;
	rTemp3: REAL;
	xRTD1Flag: BOOL;
	xRTD2Flag: BOOL;
	xRTD3Flag: BOOL;

END_VAR
VAR_OUTPUT
	END: BOOL;
	rMeasuredTemp: REAL;
	(*iFaultedRTDCount: INT;*)
END_VAR
VAR
	badRTD: INT;
	rLastMeasuredValue: REAL;
END_VAR
VAR RETAIN
END_VAR
END := FALSE;
IF EN = FALSE THEN
	RETURN;
END_IF
badRTD := BOOL_TO_INT(xRTD1Flag) + BOOL_TO_INT(xRTD2Flag) + BOOL_TO_INT(xRTD3Flag);
(*iFaultedRTDCount := badRTD;*)
CASE badRTD OF
	0:
		rMeasuredTemp := F_Median(rTemp1, rTemp2, rTemp3);
		rLastMeasuredValue := F_Median(rTemp1, rTemp2, rTemp3);
	1:
		rMeasuredTemp := F_AverageTemps(rTemp1, rTemp2, rTemp3, xRTD1Flag, xRTD2Flag, xRTD3Flag);
		rLastMeasuredValue := F_AverageTemps(rTemp1, rTemp2, rTemp3, xRTD1Flag, xRTD2Flag, xRTD3Flag);
	ELSE
		rMeasuredTemp := rLastMeasuredValue;
END_CASE
END := TRUE;
END_FUNCTION_BLOCK

(* POU Functions/F_Median, ST *)
FUNCTION F_Median : REAL
VAR_INPUT
	rValue1: REAL;
	rValue2: REAL;
	rValue3: REAL;
END_VAR
VAR
END_VAR
F_Median := MAX(MIN(rValue1, rValue2), MIN(MAX(rValue1, rValue2), rValue3));
END_FUNCTION

(* POU Functions/F_AverageTemps, ST *)
FUNCTION F_AverageTemps : REAL
VAR_INPUT
	rValue1: REAL;
	rValue2: REAL;
	rValue3: REAL;
	xTemp1Status: BOOL;
	xTemp2Status: BOOL;
	xTemp3Status: BOOL;
END_VAR
VAR
END_VAR
IF xTemp1Status = TRUE THEN
	F_AverageTemps := (rValue2 + rValue3)/2;
ELSIF xTemp2Status = TRUE THEN
	F_AverageTemps := (rValue1 + rValue3)/2;
ELSIF xTemp3Status = TRUE THEN
	F_AverageTemps := (rValue1 + rValue2)/2;
END_IF
END_FUNCTION

(* POU FB_MasterAutoTurnoverLink, ST *)
FUNCTION_BLOCK FB_MasterAutoTurnoverLink
VAR_INPUT
	EN: BOOL;
	xPrimaryAutoTurnover: BOOL;
	xSecondaryAutoTurnOver: BOOL;
END_VAR
VAR_OUTPUT
	END: BOOL;
	xMasterAutoTurnover: BOOL;
END_VAR
VAR
END_VAR
END := FALSE;
IF EN = FALSE THEN
	RETURN;
END_IF
 IF xPrimaryAutoTurnover OR xSecondaryAutoTurnOver THEN
	xMasterAutoTurnover := TRUE;
ELSE
	xMasterAutoTurnover := FALSE;
END_IF
END := TRUE;
END_FUNCTION_BLOCK

(* POU FB_FanControl, ST *)
FUNCTION_BLOCK FB_FanControl
VAR_INPUT
	EN: BOOL;
	xSystemShuttingDown: BOOL;
	xEnableFans: BOOL;
	xForceFan1On: BOOL;
	xForceFan2On: BOOL;
	xManualControl: BOOL;
END_VAR
VAR_OUTPUT
	END: BOOL;
	xCoolantFan1: BOOL;
	xCoolantFan2: BOOL;
END_VAR
VAR

END_VAR
END := FALSE;
IF EN = FALSE THEN
	RETURN;
END_IF
IF xManualControl THEN
	IF xForceFan1On AND xForceFan2On THEN
		xCoolantFan1 := TRUE;
		xCoolantFan2 := TRUE;
	ELSIF xForceFan1On AND xForceFan2On = FALSE THEN
		xCoolantFan1 := TRUE;
		xCoolantFan2 := FALSE;
	ELSIF xForceFan1On = FALSE AND xForceFan2On THEN
		xCoolantFan1 := FALSE;
		xCoolantFan2 := TRUE;
	ELSIF xForceFan1On = FALSE AND xForceFan2On = FALSE THEN
		xCoolantFan1 := FALSE;
		xCoolantFan2 := FALSE;
	END_IF
ELSIF xEnableFans = FALSE THEN
	xCoolantFan1 := FALSE;
	xCoolantFan2 := FALSE;
ELSIF xEnableFans THEN
	xCoolantFan1 := TRUE;
	xCoolantFan2 := TRUE;
END_IF

END := TRUE;
END_FUNCTION_BLOCK

(* POU FB_TemperatureController, ST *)
FUNCTION_BLOCK FB_TemperatureController
VAR_INPUT
	EN: BOOL;
	rMeasuredTemp: REAL;
	rSetpoint: REAL;
	rKp: REAL;
	rKi: REAL;
	xSystemInitializing: BOOL;
	xSystemShuttingDown: BOOL;
	xOverrideBypass: BOOL;
	SystemOn: BOOL;
END_VAR
VAR_OUTPUT
	END: BOOL;
	rOutput: REAL;
END_VAR
VAR
	rError: REAL;
	rGain: REAL := 10;
	iSample: INT := 1;
	rIntegral: REAL;
	rProportional: REAL;
END_VAR
END := FALSE;
IF EN = FALSE THEN
	RETURN;
END_IF
IF xSystemInitializing OR xSystemShuttingDown OR xOverrideBypass OR SystemOn = FALSE THEN
	rOutput := 100;
	iSample := 1;
	rIntegral := 0;
ELSE
	iSample := iSample + 1;
	rError := (rSetpoint - rMeasuredTemp);
	rIntegral := rKi * ((rIntegral + rError)/iSample);
	rProportional:= (rKp * rError);
	rOutput := rProportional + rIntegral + 50;
	IF rOutput > 100 THEN
		rOutput := 100;
	ELSIF rOutput < 0 THEN
		rOutput := 0;
	END_IF
END_IF
END := TRUE;
END_FUNCTION_BLOCK

(* POU FB_TemperatureControllerOnOff, ST *)
FUNCTION_BLOCK FB_TemperatureControllerOnOff
VAR_INPUT
	EN: BOOL;
	rMeasuredTemp: REAL;
	rLowThreshold: REAL;
	rHighThreshold: REAL;
	xSystemInitializing: BOOL;
	xSystemShuttingDown: BOOL;
	xManualControl: BOOL;
	SystemOn: BOOL;
	xForceThroughput: BOOL;
END_VAR
VAR_OUTPUT
	END: BOOL;
	rOutput: REAL;
	xEnableFans: BOOL;
END_VAR
VAR
	rError: REAL;
	rGain: REAL := 10;
	iSample: INT := 1;
	rIntegral: REAL;
	rProportional: REAL;
END_VAR
END := FALSE;
IF EN = FALSE THEN
	RETURN;
END_IF
IF xManualControl THEN
	IF xForceThroughput THEN
		rOutput := 100;
	ELSIF xForceThroughput = FALSE THEN
		rOutput := 0;
	END_IF
ELSIF xSystemInitializing OR xSystemShuttingDown OR SystemOn = FALSE THEN
	rOutput := 100;
	IF SystemOn = FALSE THEN
		xEnableFans := FALSE;
	ELSIF SystemOn = TRUE THEN
		xEnableFans := TRUE;
	END_IF
ELSIF rMeasuredTemp <= rLowThreshold THEN
	rOutput := 0;
	xEnableFans := FALSE;
ELSIF rMeasuredTemp >= rHighThreshold THEN
	rOutput := 100;
	xEnableFans := TRUE;
END_IF
END := TRUE;
END_FUNCTION_BLOCK

(* POU Legacy/FB_DigitalCapture, ST *)
FUNCTION_BLOCK FB_DigitalCapture
VAR_INPUT

	xEnable: BOOL;		(*Activates Function Block*)
	xRawInput: BOOL;
	tDebounceTime: TIME := T#50MS;		(*How long do you want to wait until it reaches a stable state*)
	xRisingEdgeDetection: BOOL; (*Is this something where we just want to measure the instance it turns on? Like user input*)
	xFallingEdgeDetection: BOOL; (*|| but off*)

END_VAR
VAR_OUTPUT
	xContinue: BOOL := TRUE;
	xRisingEdgeDetected: BOOL;
	xFallingEdgeDetected: BOOL;
END_VAR
VAR
	xRawDigitalInput: BOOL;		(*Raw Input Value from Instrument*)
	fbDebounceTimerON:TON;
	fbDebounceTimerOFF: TOF;
	fbRisingEdge: R_TRIG;
	fbFallingEdge: F_TRIG;
	iCheck: INT;
END_VAR
VAR_IN_OUT
	stInstrument: ST_INSTRUMENT;		(*User Defined Instrument*)
END_VAR
(*This takes raw digital input and stores it in instrumentation data*)
(*We need to check if 	), b) ensure hystersis does not occur (like analog), c) check if this is a user input (edge detection, versus just on/off*)

IF xEnable = FALSE THEN (*Check if we're enabled*)
	RETURN;
END_IF

(*
fbDebounceTimerON(IN := xRawInput, PT := tDebounceTime); (*Won't go to true until 50 ms of stability. Every false resets this timer*)
fbDebounceTimerOFF(IN := fbDebounceTimerON.Q, PT := tDebounceTime); (*Won't go to false until 50ms of stability. Every true resets this timer*)

xRawDigitalInput := fbDebounceTimerOFF.Q;
stInstrument.xCapturedBoolSignal := xRawDigitalInput;
fbRisingEdge(CLK := xRawDigitalInput);
fbFallingEdge(CLK := xRawDigitalInput);
IF xRisingEdgeDetection = TRUE AND xFallingEdgeDetection = TRUE THEN
	stInstrument.xCapturedBoolValue := fbRisingEdge.Q OR fbFallingEdge.Q; (*Are we detecing if this goes from False to True. When we detect this, caputre it*)
	IF (stInstrument.xCapturedBoolValue = TRUE) THEN
		iCheck := iCheck + 1;
	END_IF
ELSIF xFallingEdgeDetection = TRUE THEN
	stInstrument.xCapturedBoolValue := fbFallingEdge.Q; (*Same as above but Vice Versa. Note that you can have both!*)
	IF (stInstrument.xCapturedBoolValue = TRUE) THEN
		iCheck := iCheck + 1;
		xFallingEdgeDetected := TRUE;
	END_IF
ELSIF xRisingEdgeDetection = TRUE THEN
	stInstrument.xCapturedBoolValue := fbRisingEdge.Q;
	IF (stInstrument.xCapturedBoolValue = TRUE) THEN
		iCheck := iCheck + 1;
		xRisingEdgeDetected := TRUE;
	END_IF
ELSE
	stInstrument.xCapturedBoolValue := stInstrument.xCapturedBoolSignal;
END_IF


*)
END_FUNCTION_BLOCK

(* POU Test Bench Folder/TB_CalibrationClock, LD *)
PROGRAM TB_CalibrationClock
VAR
	a: BOOL;
	b: BOOL;
	fbct: FB_CalibrationTimer;
END_VAR
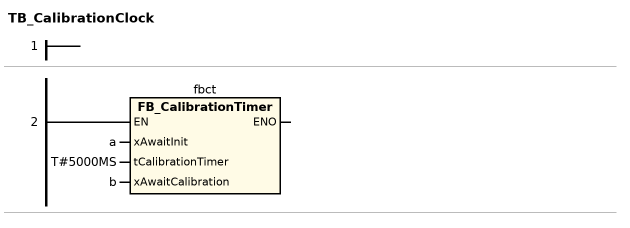
_LD_ (* Ladder Diagram *)
NETWORK 1
	*
NETWORK 2
	*
		EN --- fbct:FB_CalibrationTimer(xAwaitInit: a, tCalibrationTimer: T#5000MS, xAwaitCalibration: b)
_END_LD_
(* the same logic as Structured Text *)
(* Network 1 *)
(* Network 2 *)
fbct(xAwaitInit := a, tCalibrationTimer := T#5000MS, xAwaitCalibration := b);
END_PROGRAM

(* POU Instrument Control/Check Control/FB_CalibrationTimer, ST *)
FUNCTION_BLOCK FB_CalibrationTimer
VAR_INPUT
	xAwaitInit: BOOL;
	tCalibrationTimer: TIME;
END_VAR
VAR_OUTPUT
END_VAR
VAR
	xBeginClock: BOOL;
	fbTimerON: TON;
END_VAR
VAR_IN_OUT
	xAwaitCalibration: BOOL;
END_VAR
fbTimerON(IN := xBeginClock, PT := tCalibrationTimer);
IF xAwaitInit AND xAwaitCalibration = FALSE THEN
	xAwaitCalibration := TRUE;
ELSIF xAwaitInit = FALSE AND (xAwaitCalibration OR xBeginClock) THEN
	xBeginClock := TRUE;
ELSIF xAwaitInit AND xBeginClock THEN
	xBeginClock := FALSE;
	xAwaitCalibration := TRUE;
ELSIF xAwaitInit AND xAwaitCalibration THEN
	RETURN;
END_IF

IF xBeginClock = TRUE AND fbTimerON.Q = TRUE THEN
	xAwaitCalibration := FALSE;
	xBeginClock := FALSE;
END_IF
END_FUNCTION_BLOCK

(* POU Test Bench Folder/TB_CheckConductivity, LD *)
PROGRAM TB_CheckConductivity
VAR
	a: BOOL := FALSE;
	b: BOOL := FALSE;
	c: BOOL := FALSE;
	d: REAL := 4;
	e: REAL := 10;
	f: REAL := 15;
	z: BOOL;
	y: BOOL;
	x: BOOL;
	w: BOOL;
	v: BOOL;
	u: BOOL;
	fbcc: FB_CheckConductivity;
END_VAR
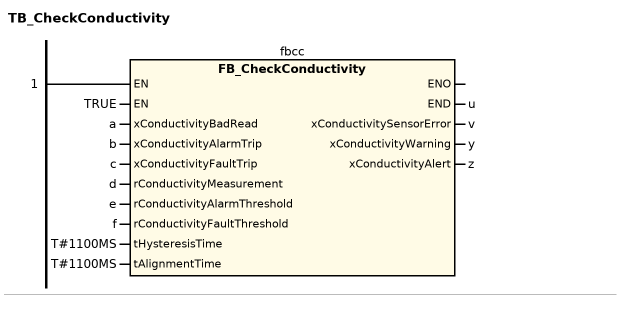
_LD_ (* Ladder Diagram *)
NETWORK 1
	*
		EN --- fbcc:FB_CheckConductivity(EN: TRUE, xConductivityBadRead: a, xConductivityAlarmTrip: b, xConductivityFaultTrip: c, rConductivityMeasurement: d, rConductivityAlarmThreshold: e, rConductivityFaultThreshold: f, tHysteresisTime: T#1100MS, tAlignmentTime: T#1100MS, xConductivitySensorError => v, xConductivityWarning => y, xConductivityAlert => z) => u
_END_LD_
(* the same logic as Structured Text *)
(* Network 1 *)
fbcc(EN := TRUE, xConductivityBadRead := a, xConductivityAlarmTrip := b, xConductivityFaultTrip := c, rConductivityMeasurement := d, rConductivityAlarmThreshold := e, rConductivityFaultThreshold := f, tHysteresisTime := T#1100MS, tAlignmentTime := T#1100MS);
v := fbcc.xConductivitySensorError;
y := fbcc.xConductivityWarning;
z := fbcc.xConductivityAlert;
u := fbcc.END;
END_PROGRAM

(* POU Test Bench Folder/TB_InputTest, LD *)
PROGRAM TB_InputTest
VAR
	xOnOff: BOOL;
END_VAR
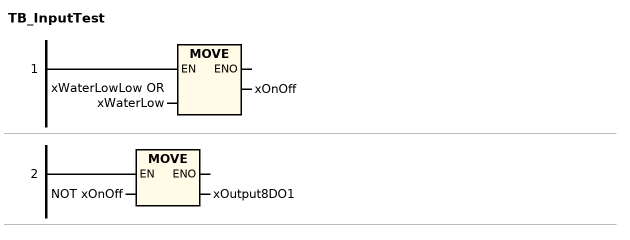
_LD_ (* Ladder Diagram *)
NETWORK 1
	*
		EN --- MOVE( xWaterLowLow OR xWaterLow) => xOnOff
NETWORK 2
	*
		EN --- MOVE(NOT xOnOff) => xOutput8DO1
_END_LD_
(* the same logic as Structured Text *)
(* Network 1 *)
xOnOff :=  xWaterLowLow OR xWaterLow;
(* Network 2 *)
xOutput8DO1 := NOT xOnOff;
END_PROGRAM

(* POU Test Bench Folder/TB_InstrumentReadErrorFaultAlignment, LD *)
PROGRAM TB_InstrumentReadErrorFaultAlignment
VAR
	pbr1: BOOL := FALSE;
	pbr2: BOOL := FALSE;
	tbr1: BOOL := FALSE;
	tbr2: BOOL := FALSE;
	tbr3: BOOL := FALSE;
	cbr: BOOL := FALSE;
	fbr: BOOL := FALSE;
	pef1: BOOL;
	pef2: BOOL;
	pef3: BOOL;
	tef1: BOOL;
	tef2: BOOL;
	tef3: BOOL;
	cef: BOOL;
	fef: BOOL;
	fbirr: FB_InstrumentReadRecon;
END_VAR
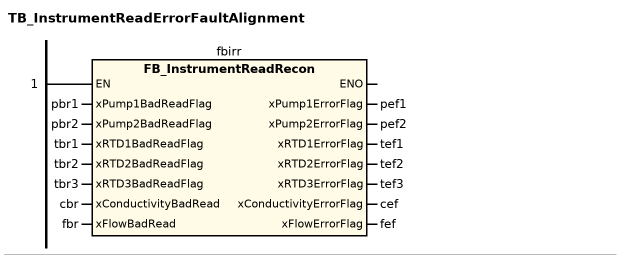
_LD_ (* Ladder Diagram *)
NETWORK 1
	*
		EN --- fbirr:FB_InstrumentReadRecon(xPump1BadReadFlag: pbr1, xPump2BadReadFlag: pbr2, xRTD1BadReadFlag: tbr1, xRTD2BadReadFlag: tbr2, xRTD3BadReadFlag: tbr3, xConductivityBadRead: cbr, xFlowBadRead: fbr, xPump2ErrorFlag => pef2, xRTD1ErrorFlag => tef1, xRTD2ErrorFlag => tef2, xRTD3ErrorFlag => tef3, xConductivityErrorFlag => cef, xFlowErrorFlag => fef) => pef1
_END_LD_
(* the same logic as Structured Text *)
(* Network 1 *)
fbirr(xPump1BadReadFlag := pbr1, xPump2BadReadFlag := pbr2, xRTD1BadReadFlag := tbr1, xRTD2BadReadFlag := tbr2, xRTD3BadReadFlag := tbr3, xConductivityBadRead := cbr, xFlowBadRead := fbr);
pef2 := fbirr.xPump2ErrorFlag;
tef1 := fbirr.xRTD1ErrorFlag;
tef2 := fbirr.xRTD2ErrorFlag;
tef3 := fbirr.xRTD3ErrorFlag;
cef := fbirr.xConductivityErrorFlag;
fef := fbirr.xFlowErrorFlag;
pef1 := fbirr.xPump1ErrorFlag;
END_PROGRAM

(* POU Data Conversion/Instrument->System/FB_InstrumentReadRecon, ST *)
FUNCTION_BLOCK FB_InstrumentReadRecon
VAR_INPUT
	xPump1BadReadFlag: BOOL;
	xPump2BadReadFlag: BOOL;
	xRTD1BadReadFlag: BOOL;
	xRTD2BadReadFlag: BOOL;
	xRTD3BadReadFlag: BOOL;
	xConductivityBadRead: BOOL;
	xFlowBadRead: BOOL;
END_VAR
VAR_OUTPUT
	xPump1ErrorFlag: BOOL;
	xPump2ErrorFlag: BOOL;
	xRTD1ErrorFlag: BOOL;
	xRTD2ErrorFlag: BOOL;
	xRTD3ErrorFlag: BOOL;
	xConductivityErrorFlag: BOOL;
	xFlowErrorFlag: BOOL;
END_VAR
VAR
END_VAR
 xPump1ErrorFlag :=  xPump1BadReadFlag;
xPump2ErrorFlag := xPump2BadReadFlag;
xRTD1ErrorFlag := xRTD1BadReadFlag;
xRTD2ErrorFlag :=  xRTD2BadReadFlag;
xRTD3ErrorFlag := xRTD3BadReadFlag;
 xConductivityErrorFlag := xConductivityBadRead;
xFlowErrorFlag := xFlowBadRead;
END_FUNCTION_BLOCK

(* POU Test Bench Folder/TB_PowerPressureFlowVote, LD *)
PROGRAM TB_PowerPressureFlowVote
VAR

	fbppfv: FB_PowerPressureFlowVote;
	fbpssr: FB_PumpStartSwitchRoutine;
	p1ff: BOOL;
	p2ff: BOOL;
	p1lpf: BOOL;
	p2lpf: BOOL;
	nbf: BOOL;
	rpsf: BOOL;
	awif: BOOL;
	sysp1o: BOOL;
	sysp2o: BOOL;
	sysa: BOOL;
	sysf: BOOL;
	syspp: REAL := 15;
	sysppl: BOOL;
	sysfl: BOOL;
	syspl: BOOL;
	active: INT := 1;
	fbppft: FB_PowerPressureFlowThreshold;
	pressure: BOOL := TRUE;
END_VAR
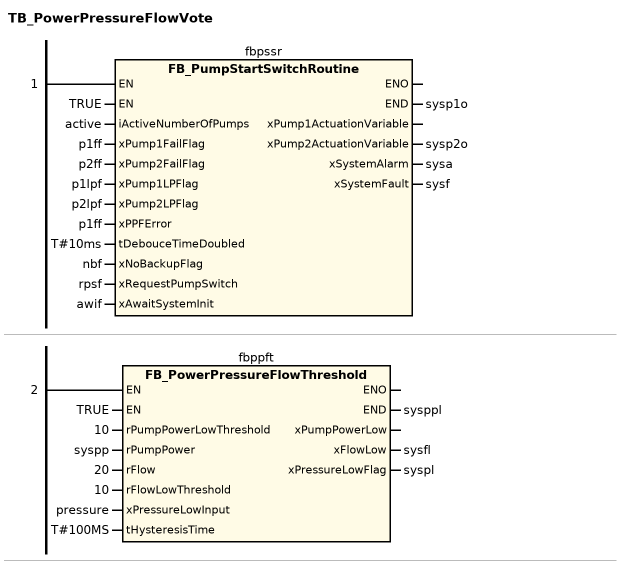
_LD_ (* Ladder Diagram *)
NETWORK 1
	*
		EN --- fbpssr:FB_PumpStartSwitchRoutine(EN: TRUE, iActiveNumberOfPumps: active, xPump1FailFlag: p1ff, xPump2FailFlag: p2ff, xPump1LPFlag: p1lpf, xPump2LPFlag: p2lpf, xPPFError: p1ff, tDebouceTimeDoubled: T#10ms, xNoBackupFlag: nbf, xRequestPumpSwitch: rpsf, xAwaitSystemInit: awif, xPump2ActuationVariable => sysp2o, xSystemAlarm => sysa, xSystemFault => sysf) => sysp1o
NETWORK 2
	*
		EN --- fbppft:FB_PowerPressureFlowThreshold(EN: TRUE, rPumpPowerLowThreshold: 10, rPumpPower: syspp, rFlow: 20, rFlowLowThreshold: 10, xPressureLowInput: pressure, tHysteresisTime: T#100MS, xFlowLow => sysfl, xPressureLowFlag => syspl) => sysppl
_END_LD_
(* the same logic as Structured Text *)
(* Network 1 *)
fbpssr(EN := TRUE, iActiveNumberOfPumps := active, xPump1FailFlag := p1ff, xPump2FailFlag := p2ff, xPump1LPFlag := p1lpf, xPump2LPFlag := p2lpf, xPPFError := p1ff, tDebouceTimeDoubled := T#10ms, xNoBackupFlag := nbf, xRequestPumpSwitch := rpsf, xAwaitSystemInit := awif);
sysp2o := fbpssr.xPump2ActuationVariable;
sysa := fbpssr.xSystemAlarm;
sysf := fbpssr.xSystemFault;
sysp1o := fbpssr.END;
(* Network 2 *)
fbppft(EN := TRUE, rPumpPowerLowThreshold := 10, rPumpPower := syspp, rFlow := 20, rFlowLowThreshold := 10, xPressureLowInput := pressure, tHysteresisTime := T#100MS);
sysfl := fbppft.xFlowLow;
syspl := fbppft.xPressureLowFlag;
sysppl := fbppft.END;
END_PROGRAM

(* POU Instrument Control/FB_PumpStartSwitchRoutine, ST *)
FUNCTION_BLOCK FB_PumpStartSwitchRoutine
VAR_INPUT
	EN: BOOL;
	iActiveNumberOfPumps: INT;
	xPump1FailFlag: BOOL;
	xPump2FailFlag: BOOL;
	xPump1LPFlag: BOOL;
	xPump2LPFlag: BOOL;
	xPPFError: BOOL;
	tDebouceTimeDoubled: TIME;
END_VAR
VAR_OUTPUT
	END: BOOL;
	xPump1ActuationVariable: BOOL;
	xPump2ActuationVariable: BOOL;
	xSystemAlarm: BOOL;
	xSystemFault: BOOL;
END_VAR
VAR
	fbbypass: TON;
END_VAR
VAR_IN_OUT
	xNoBackupFlag: BOOL;
	xRequestPumpSwitch: BOOL;
	xAwaitSystemInit: BOOL;
END_VAR
fbbypass(IN := TRUE,  PT := tDebouceTimeDoubled);
IF EN = FALSE OR fbbypass.Q = FALSE  THEN
	RETURN;
END_IF
END := FALSE;
IF xRequestPumpSwitch AND xNoBackupFlag THEN
	xSystemFault := TRUE;
	xPump1ActuationVariable := FALSE;
	xPump2ActuationVariable := FALSE;
ELSIF xRequestPumpSwitch AND xNoBackupFlag = FALSE AND xAwaitSystemInit = FALSE THEN
	xAwaitSystemInit := TRUE;
	CASE  iActiveNumberOfPumps OF
		0:
			IF (xPump1FailFlag OR xPump1LPFlag) THEN
				xPump1ActuationVariable := FALSE;
				xPump2ActuationVariable := TRUE;
			ELSIF (xPump1FailFlag = FALSE OR xPump1LPFlag = FALSE) THEN
				xPump1ActuationVariable := TRUE;
				xPump2ActuationVariable := FALSE;
			END_IF
		1:
			xPump1ActuationVariable := FALSE;
			xPump2ActuationVariable := TRUE;
			IF (xPump1FailFlag OR (xPump1LPFlag AND xPPFError)) THEN
				xNoBackupFlag := TRUE;
				xSystemAlarm := TRUE;
			END_IF
		2:
			xPump1ActuationVariable := TRUE;
			xPump2ActuationVariable := FALSE;
			IF (xPump2FailFlag OR (xPump2LPFlag AND xPPFError)) THEN
				xNoBackupFlag := TRUE;
				xSystemAlarm := TRUE;
			END_IF
		ELSE
			xSystemFault := TRUE;
			xPump1ActuationVariable := FALSE;
			xPump2ActuationVariable := FALSE;
			xNoBackupFlag := TRUE;
	END_CASE
END_IF
xRequestPumpSwitch := FALSE;
END := TRUE;
END_FUNCTION_BLOCK

(* POU Test Bench Folder/TB_SystemInstrumentAlignment, LD *)
PROGRAM TB_SystemInstrumentAlignment
VAR
	pump1: ST_INSTRUMENT;
	pump2: ST_INSTRUMENT;
	temp1: ST_INSTRUMENT;
	temp2: ST_INSTRUMENT;
	temp3: ST_INSTRUMENT;
	flow: ST_INSTRUMENT;
	pressure: ST_INSTRUMENT;
	conduct: ST_INSTRUMENT;
	low: ST_INSTRUMENT;
	lowlow: ST_INSTRUMENT;
	sys: ST_SYSTEM;
	fbsia: FB_SystemInstrumentAlignment;
	flags: ST_InstrumentFlags;
	xa: BOOL := FALSE;
	xb: BOOL := FALSE;
	t1: BOOL := FALSE;
	t2: BOOL := FALSE;
	t3: BOOL := FALSE;
	c1: BOOL := FALSE;
	f1: BOOL := FALSE;
END_VAR
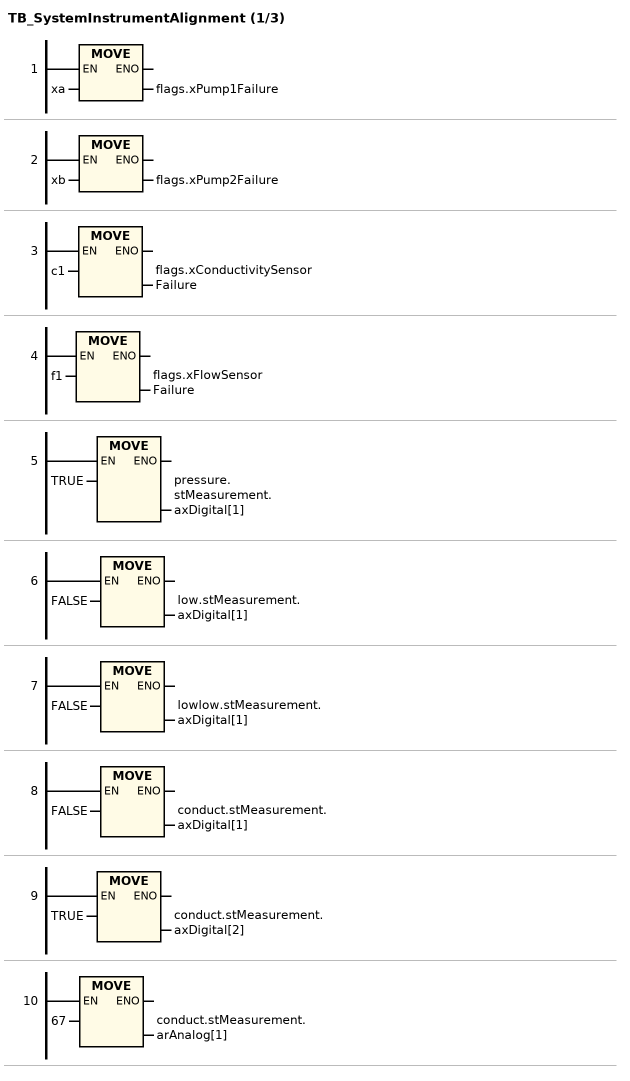
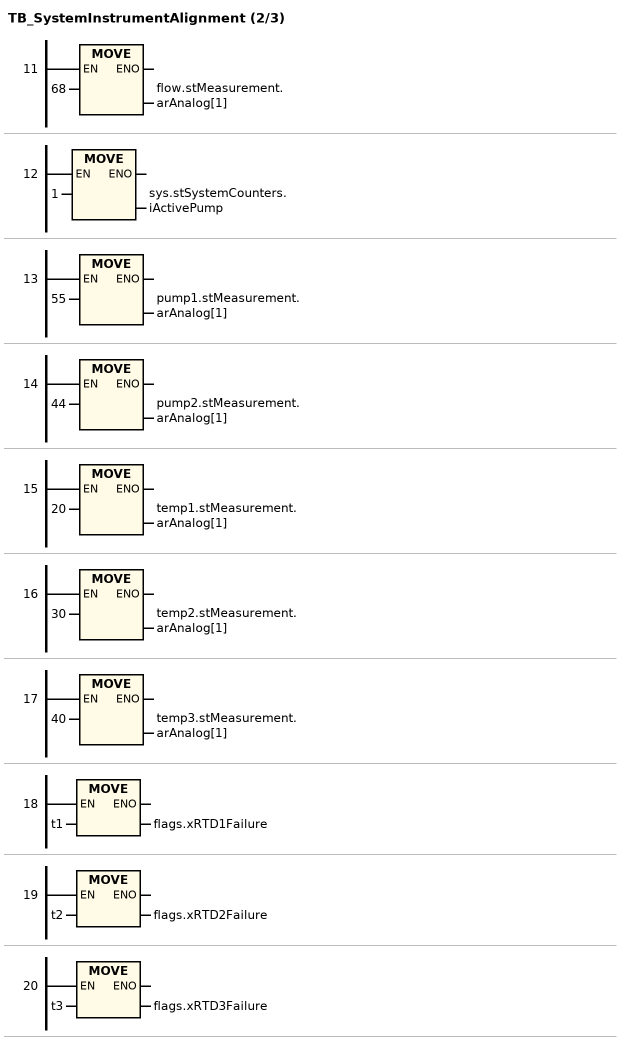
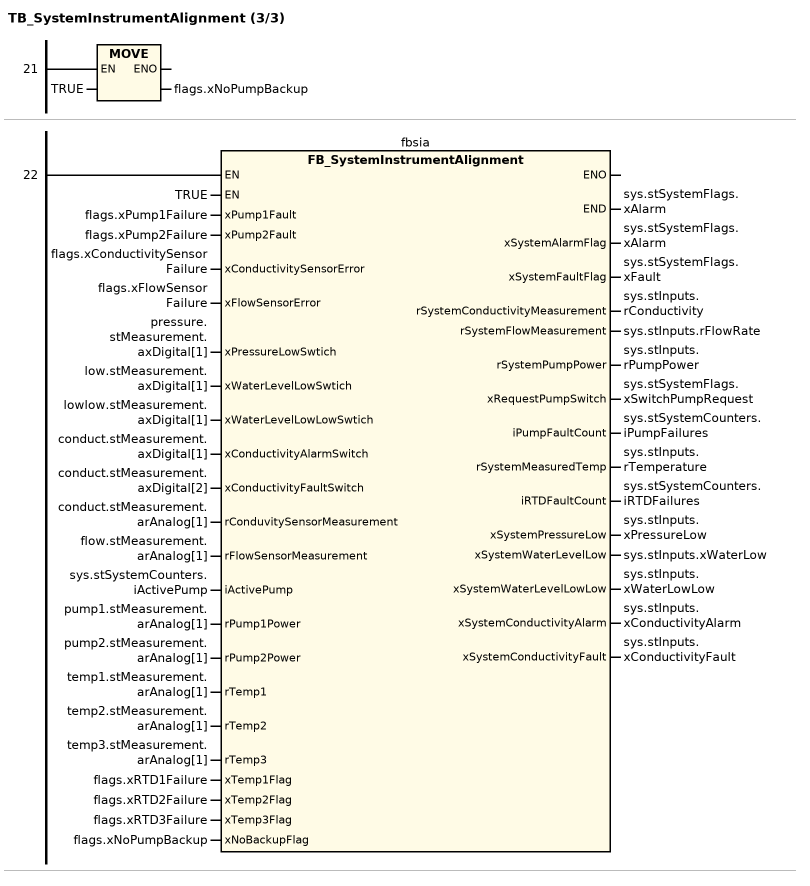
_LD_ (* Ladder Diagram *)
NETWORK 1
	*
		EN --- MOVE(xa) => flags.xPump1Failure
NETWORK 2
	*
		EN --- MOVE(xb) => flags.xPump2Failure
NETWORK 3
	*
		EN --- MOVE(c1) => flags.xConductivitySensorFailure
NETWORK 4
	*
		EN --- MOVE(f1) => flags.xFlowSensorFailure
NETWORK 5
	*
		EN --- MOVE(TRUE) => pressure.stMeasurement.axDigital[1]
NETWORK 6
	*
		EN --- MOVE(FALSE) => low.stMeasurement.axDigital[1]
NETWORK 7
	*
		EN --- MOVE(FALSE) => lowlow.stMeasurement.axDigital[1]
NETWORK 8
	*
		EN --- MOVE(FALSE) => conduct.stMeasurement.axDigital[1]
NETWORK 9
	*
		EN --- MOVE(TRUE) => conduct.stMeasurement.axDigital[2]
NETWORK 10
	*
		EN --- MOVE(67) => conduct.stMeasurement.arAnalog[1]
NETWORK 11
	*
		EN --- MOVE(68) => flow.stMeasurement.arAnalog[1]
NETWORK 12
	*
		EN --- MOVE(1) => sys.stSystemCounters.iActivePump
NETWORK 13
	*
		EN --- MOVE(55) => pump1.stMeasurement.arAnalog[1]
NETWORK 14
	*
		EN --- MOVE(44) => pump2.stMeasurement.arAnalog[1]
NETWORK 15
	*
		EN --- MOVE(20) => temp1.stMeasurement.arAnalog[1]
NETWORK 16
	*
		EN --- MOVE(30) => temp2.stMeasurement.arAnalog[1]
NETWORK 17
	*
		EN --- MOVE(40) => temp3.stMeasurement.arAnalog[1]
NETWORK 18
	*
		EN --- MOVE(t1) => flags.xRTD1Failure
NETWORK 19
	*
		EN --- MOVE(t2) => flags.xRTD2Failure
NETWORK 20
	*
		EN --- MOVE(t3) => flags.xRTD3Failure
NETWORK 21
	*
		EN --- MOVE(TRUE) => flags.xNoPumpBackup
NETWORK 22
	*
		EN --- fbsia:FB_SystemInstrumentAlignment(EN: TRUE, xPump1Fault: flags.xPump1Failure, xPump2Fault: flags.xPump2Failure, xConductivitySensorError: flags.xConductivitySensorFailure, xFlowSensorError: flags.xFlowSensorFailure, xPressureLowSwtich: pressure.stMeasurement.axDigital[1], xWaterLevelLowSwtich: low.stMeasurement.axDigital[1], xWaterLevelLowLowSwtich: lowlow.stMeasurement.axDigital[1], xConductivityAlarmSwitch: conduct.stMeasurement.axDigital[1], xConductivityFaultSwitch: conduct.stMeasurement.axDigital[2], rConduvitySensorMeasurement: conduct.stMeasurement.arAnalog[1], rFlowSensorMeasurement: flow.stMeasurement.arAnalog[1], iActivePump: sys.stSystemCounters.iActivePump, rPump1Power: pump1.stMeasurement.arAnalog[1], rPump2Power: pump2.stMeasurement.arAnalog[1], rTemp1: temp1.stMeasurement.arAnalog[1], rTemp2: temp2.stMeasurement.arAnalog[1], rTemp3: temp3.stMeasurement.arAnalog[1], xTemp1Flag: flags.xRTD1Failure, xTemp2Flag: flags.xRTD2Failure, xTemp3Flag: flags.xRTD3Failure, xNoBackupFlag: flags.xNoPumpBackup, xSystemAlarmFlag => sys.stSystemFlags.xAlarm, xSystemFaultFlag => sys.stSystemFlags.xFault, rSystemConductivityMeasurement => sys.stInputs.rConductivity, rSystemFlowMeasurement => sys.stInputs.rFlowRate, rSystemPumpPower => sys.stInputs.rPumpPower, xRequestPumpSwitch => sys.stSystemFlags.xSwitchPumpRequest, iPumpFaultCount => sys.stSystemCounters.iPumpFailures, rSystemMeasuredTemp => sys.stInputs.rTemperature, iRTDFaultCount => sys.stSystemCounters.iRTDFailures, xSystemPressureLow => sys.stInputs.xPressureLow, xSystemWaterLevelLow => sys.stInputs.xWaterLow, xSystemWaterLevelLowLow => sys.stInputs.xWaterLowLow, xSystemConductivityAlarm => sys.stInputs.xConductivityAlarm, xSystemConductivityFault => sys.stInputs.xConductivityFault) => sys.stSystemFlags.xAlarm
_END_LD_
(* the same logic as Structured Text *)
(* Network 1 *)
flags.xPump1Failure := xa;
(* Network 2 *)
flags.xPump2Failure := xb;
(* Network 3 *)
flags.xConductivitySensorFailure := c1;
(* Network 4 *)
flags.xFlowSensorFailure := f1;
(* Network 5 *)
pressure.stMeasurement.axDigital[1] := TRUE;
(* Network 6 *)
low.stMeasurement.axDigital[1] := FALSE;
(* Network 7 *)
lowlow.stMeasurement.axDigital[1] := FALSE;
(* Network 8 *)
conduct.stMeasurement.axDigital[1] := FALSE;
(* Network 9 *)
conduct.stMeasurement.axDigital[2] := TRUE;
(* Network 10 *)
conduct.stMeasurement.arAnalog[1] := 67;
(* Network 11 *)
flow.stMeasurement.arAnalog[1] := 68;
(* Network 12 *)
sys.stSystemCounters.iActivePump := 1;
(* Network 13 *)
pump1.stMeasurement.arAnalog[1] := 55;
(* Network 14 *)
pump2.stMeasurement.arAnalog[1] := 44;
(* Network 15 *)
temp1.stMeasurement.arAnalog[1] := 20;
(* Network 16 *)
temp2.stMeasurement.arAnalog[1] := 30;
(* Network 17 *)
temp3.stMeasurement.arAnalog[1] := 40;
(* Network 18 *)
flags.xRTD1Failure := t1;
(* Network 19 *)
flags.xRTD2Failure := t2;
(* Network 20 *)
flags.xRTD3Failure := t3;
(* Network 21 *)
flags.xNoPumpBackup := TRUE;
(* Network 22: see the listing above *)
END_PROGRAM

(* POU Data Conversion/Instrument->System/FB_SystemInstrumentAlignment, LD *)
FUNCTION_BLOCK FB_SystemInstrumentAlignment
VAR_INPUT
	EN: BOOL;
	xPump1Fault: BOOL;
	xPump2Fault: BOOL;
	xConductivitySensorError: BOOL;
	xFlowSensorError: BOOL;
	xPressureLowSwtich: BOOL;
	xWaterLevelLowSwtich: BOOL;
	xWaterLevelLowLowSwtich: BOOL;
	xConductivityAlarmSwitch: BOOL;
	xConductivityFaultSwitch: BOOL;
	rConduvitySensorMeasurement: REAL;
	rFlowSensorMeasurement: REAL;
	iActivePump: INT;
	rPump1Power: REAL;
	rPump2Power: REAL;
	rTemp1: REAL;
	rTemp2: REAL;
	rTemp3: REAL;
	xTemp1Flag: BOOL;
	xTemp2Flag: BOOL;
	xTemp3Flag: BOOL;

END_VAR
VAR_OUTPUT
	END: BOOL;
	xSystemAlarmFlag: BOOL;
	xSystemFaultFlag: BOOL;
	rSystemConductivityMeasurement: REAL;
	rSystemFlowMeasurement: REAL;
	rSystemPumpPower: REAL;
	xRequestPumpSwitch: BOOL;
	iPumpFaultCount: INT;
	rSystemMeasuredTemp: REAL;
	iRTDFaultCount: INT;
	xSystemPressureLow: BOOL;
	xSystemWaterLevelLow: BOOL;
	xSystemWaterLevelLowLow: BOOL;
	xSystemConductivityAlarm: BOOL;
	xSystemConductivityFault: BOOL;

END_VAR
VAR
	fbcfsa: FB_CondFlowSystemAlignment;
	fbcfsa2: FB_CondFlowSystemAlignment;
	fbpsa: FB_PumpSystemAlignment;

	fbtsa: FB_TempSystemAlignment;

	xSystemFaultFlag1: BOOL;
	xSystemFaultFlag2: BOOL;
	xSystemFaultFlag3: BOOL;
	xSystemFaultFlag4: BOOL;
	xSystemAlarmFlag1: BOOL;
	xSystemAlarmFlag2: BOOL;
	xSystemAlarmFlag3: BOOL;
	xSAFcontact: BOOL;
	xSAAcontact: BOOL;
END_VAR
VAR_IN_OUT
	xNoBackupFlag: BOOL;

END_VAR
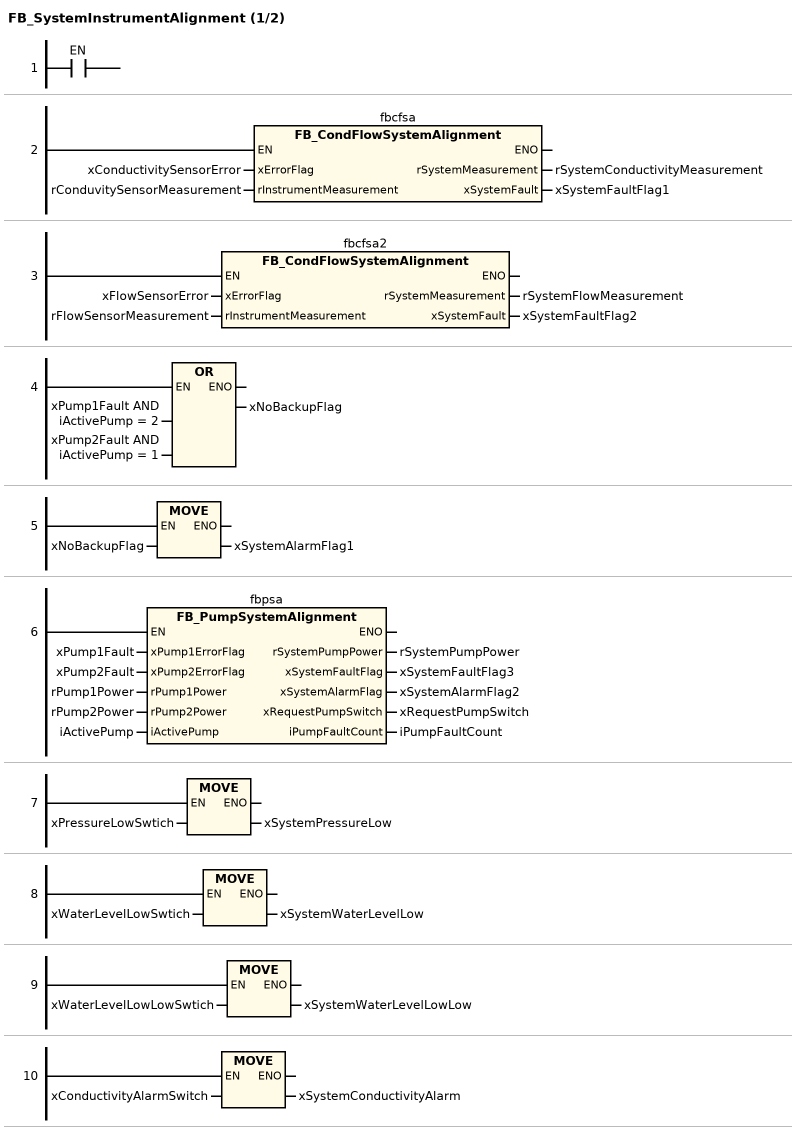
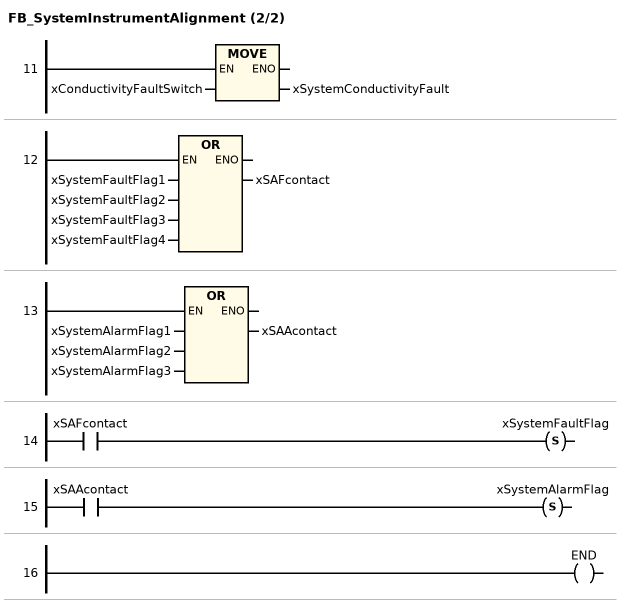
_LD_ (* Ladder Diagram *)
NETWORK 1
	[EN]
NETWORK 2
	*
		EN --- fbcfsa:FB_CondFlowSystemAlignment(xErrorFlag: xConductivitySensorError, rInstrumentMeasurement: rConduvitySensorMeasurement, xSystemFault => xSystemFaultFlag1) => rSystemConductivityMeasurement
NETWORK 3
	*
		EN --- fbcfsa2:FB_CondFlowSystemAlignment(xErrorFlag: xFlowSensorError, rInstrumentMeasurement: rFlowSensorMeasurement, xSystemFault => xSystemFaultFlag2) => rSystemFlowMeasurement
NETWORK 4
	*
		EN --- OR(xPump1Fault AND iActivePump = 2, xPump2Fault AND iActivePump = 1) => xNoBackupFlag
NETWORK 5
	*
		EN --- MOVE(xNoBackupFlag) => xSystemAlarmFlag1
NETWORK 6
	*
		EN --- fbpsa:FB_PumpSystemAlignment(xPump1ErrorFlag: xPump1Fault, xPump2ErrorFlag: xPump2Fault, rPump1Power: rPump1Power, rPump2Power: rPump2Power, iActivePump: iActivePump, xSystemFaultFlag => xSystemFaultFlag3, xSystemAlarmFlag => xSystemAlarmFlag2, xRequestPumpSwitch => xRequestPumpSwitch, iPumpFaultCount => iPumpFaultCount) => rSystemPumpPower
NETWORK 7
	*
		EN --- MOVE(xPressureLowSwtich) => xSystemPressureLow
NETWORK 8
	*
		EN --- MOVE(xWaterLevelLowSwtich) => xSystemWaterLevelLow
NETWORK 9
	*
		EN --- MOVE(xWaterLevelLowLowSwtich) => xSystemWaterLevelLowLow
NETWORK 10
	*
		EN --- MOVE(xConductivityAlarmSwitch) => xSystemConductivityAlarm
NETWORK 11
	*
		EN --- MOVE(xConductivityFaultSwitch) => xSystemConductivityFault
NETWORK 12
	*
		EN --- OR(xSystemFaultFlag1, xSystemFaultFlag2, xSystemFaultFlag3, xSystemFaultFlag4) => xSAFcontact
NETWORK 13
	*
		EN --- OR(xSystemAlarmFlag1, xSystemAlarmFlag2, xSystemAlarmFlag3) => xSAAcontact
NETWORK 14
	[xSAFcontact] --- (S xSystemFaultFlag)
NETWORK 15
	[xSAAcontact] --- (S xSystemAlarmFlag)
NETWORK 16
	* --- (END)
_END_LD_
(* the same logic as Structured Text *)
(* Network 1 *)
(* Network 2 *)
fbcfsa(xErrorFlag := xConductivitySensorError, rInstrumentMeasurement := rConduvitySensorMeasurement);
xSystemFaultFlag1 := fbcfsa.xSystemFault;
rSystemConductivityMeasurement := fbcfsa.rSystemMeasurement;
(* Network 3 *)
fbcfsa2(xErrorFlag := xFlowSensorError, rInstrumentMeasurement := rFlowSensorMeasurement);
xSystemFaultFlag2 := fbcfsa2.xSystemFault;
rSystemFlowMeasurement := fbcfsa2.rSystemMeasurement;
(* Network 4 *)
xNoBackupFlag := (xPump1Fault AND iActivePump = 2) OR (xPump2Fault AND iActivePump = 1);
(* Network 5 *)
xSystemAlarmFlag1 := xNoBackupFlag;
(* Network 6 *)
fbpsa(xPump1ErrorFlag := xPump1Fault, xPump2ErrorFlag := xPump2Fault, rPump1Power := rPump1Power, rPump2Power := rPump2Power, iActivePump := iActivePump);
xSystemFaultFlag3 := fbpsa.xSystemFaultFlag;
xSystemAlarmFlag2 := fbpsa.xSystemAlarmFlag;
xRequestPumpSwitch := fbpsa.xRequestPumpSwitch;
iPumpFaultCount := fbpsa.iPumpFaultCount;
rSystemPumpPower := fbpsa.rSystemPumpPower;
(* Network 7 *)
xSystemPressureLow := xPressureLowSwtich;
(* Network 8 *)
xSystemWaterLevelLow := xWaterLevelLowSwtich;
(* Network 9 *)
xSystemWaterLevelLowLow := xWaterLevelLowLowSwtich;
(* Network 10 *)
xSystemConductivityAlarm := xConductivityAlarmSwitch;
(* Network 11 *)
xSystemConductivityFault := xConductivityFaultSwitch;
(* Network 12 *)
xSAFcontact := xSystemFaultFlag1 OR xSystemFaultFlag2 OR xSystemFaultFlag3 OR xSystemFaultFlag4;
(* Network 13 *)
xSAAcontact := xSystemAlarmFlag1 OR xSystemAlarmFlag2 OR xSystemAlarmFlag3;
(* Network 14 *)
IF xSAFcontact THEN xSystemFaultFlag := TRUE; END_IF;
(* Network 15 *)
IF xSAAcontact THEN xSystemAlarmFlag := TRUE; END_IF;
(* Network 16 *)
END := TRUE;
END_FUNCTION_BLOCK

(* POU Data Conversion/Instrument->System/FB_CondFlowSystemAlignment, ST *)
FUNCTION_BLOCK FB_CondFlowSystemAlignment
VAR_INPUT
	xErrorFlag: BOOL;
	rInstrumentMeasurement: REAL;
END_VAR
VAR_OUTPUT
	rSystemMeasurement: REAL;
	xSystemFault: BOOL;
END_VAR
VAR
	rLastRead: REAL := 0;
END_VAR
IF xErrorFlag = TRUE THEN
	rSystemMeasurement := rLastRead;
	xSystemFault := TRUE;
ELSE
	rSystemMeasurement := rInstrumentMeasurement;
	rLastRead := rInstrumentMeasurement;
END_IF
END_FUNCTION_BLOCK

(* POU Data Conversion/Instrument->System/FB_PumpSystemAlignment, ST *)
FUNCTION_BLOCK FB_PumpSystemAlignment
VAR_INPUT

	xPump1ErrorFlag: BOOL;
	xPump2ErrorFlag: BOOL;
	rPump1Power: REAL;
	rPump2Power: REAL;
	iActivePump: INT;
END_VAR
VAR_OUTPUT
	rSystemPumpPower: REAL;

	xSystemFaultFlag: BOOL;
	xSystemAlarmFlag: BOOL;
	xRequestPumpSwitch: BOOL;
	iPumpFaultCount: INT;
END_VAR
VAR
	rLastPumpPowerRead: REAL;
END_VAR
VAR_IN_OUT

END_VAR
iPumpFaultCount := BOOL_TO_INT(xPump1ErrorFlag) + BOOL_TO_INT(xPump2ErrorFlag);
IF (xPump1ErrorFlag AND xPump2ErrorFlag) THEN
	xSystemFaultFlag := TRUE;
	xRequestPumpSwitch := TRUE;
ELSIF (xPump1ErrorFlag AND iActivePump = 1) OR (xPump2ErrorFlag AND iActivePump = 2) THEN
	rSystemPumpPower := rLastPumpPowerRead;
	xSystemAlarmFlag := TRUE;
	xRequestPumpSwitch := TRUE;
ELSIF iActivePump = 0 THEN
	xRequestPumpSwitch := TRUE;
	rSystemPumpPower := 0;
ELSIF iActivePump = 1 THEN
	rLastPumpPowerRead := rSystemPumpPower;
	rSystemPumpPower := rPump1Power;
ELSIF iActivePump = 2 THEN
	rLastPumpPowerRead := rSystemPumpPower;
	rSystemPumpPower := rPump2Power;
	END_IF
END_FUNCTION_BLOCK

(* POU Legacy/TB_TempValCtrlSys, ST *)
PROGRAM TB_TempValCtrlSys
VAR
	temp1Val: REAL;
	temp2Val: REAL;
	temp3Val: REAL;
	temp1Alarm: BOOL;
	temp2Alarm: BOOL;
	temp3Aalrm: BOOL;
	temp1Fault: BOOL;
	temp2Fault: BOOL;
	temp3Fault: BOOL;
	threshold: REAL;
	tolearnce: REAL;
	ctrlAlarm: BOOL;
	ctrlFault: BOOL;
	pgrmError: BOOL;
	UUT: FB_TempValCtrlSys;
END_VAR
temp1Val :=  gaTemps[1].stTempRead.rProcessed;
temp2Val := gaTemps[2].stTempRead.rProcessed;
	temp3Val := gaTemps[3].stTempRead.rProcessed;
	temp1Alarm := gaTemps[1].stDescription.xAlarm;
	temp2Alarm := gaTemps[2].stDescription.xAlarm;
	temp3Aalrm := gaTemps[3].stDescription.xAlarm;
	temp1Fault := gaTemps[1].stDescription.xFault;
	temp2Fault := gaTemps[2].stDescription.xFault;
	temp3Fault := gaTemps[3].stDescription.xFault;
	threshold := gTempValCtrlSys.rDiffThresh;
	tolearnce := gTempValCtrlSys.rDiffTol;
	ctrlAlarm := gTempValCtrlSys.xAlarm;
	ctrlFault := gTempValCtrlSys.xFault;
	pgrmError := gProgramErrors.xTempValCtrlSys;

gaTemps[1].stTempRead.rProcessed := 0;
gaTemps[2].stTempRead.rProcessed := 0;
gaTemps[3].stTempRead.rProcessed := 0;
gaTemps[1].stDescription.xAlarm := FALSE;
gaTemps[2].stDescription.xAlarm := FALSE;
gaTemps[3].stDescription.xAlarm := FALSE;
gaTemps[1].stDescription.xFault := FALSE;
gaTemps[2].stDescription.xFault := FALSE;
gaTemps[3].stDescription.xFault := FALSE;
gTempValCtrlSys.rDiffThresh := 0;
gTempValCtrlSys.rDiffTol := 0;
gTempValCtrlSys.xAlarm := FALSE;
gTempValCtrlSys.xFault := FALSE;
gProgramErrors.xTempValCtrlSys := FALSE;

gaTemps[1].stTempRead.rProcessed := -1;
gaTemps[2].stTempRead.rProcessed := 0;
gaTemps[3].stTempRead.rProcessed := 1;
gTempValCtrlSys.rDiffThresh := 30;
gTempValCtrlSys.rDiffTol := 10;
UUT();
(*
CASE iTestStep OF
	0: (* Initialize Function*)
		SET(
	xTempAlarm: ARRAY [1..3] OF BOOL;
	xCtrlSysFault: BOOL;
	xCtrlSysAlarm: BOOL;
		UUT();
		tbTBLog := CONCAT(tbTBLog, 'S');
		iTestStep := iTestStep + 1;
	1:
		gaTemps[1].stDescription.xFault:= 5;
		gaTemps[2].stTempRead.rProcessed := 5;
		gaTemps[3].stTempRead.rProcessed := 5
		tbTBLog := CONCAT(tbTBLog, '1');
		FOR i := 1 TO 2 DO
			gaPumps[i].stPumpPower.iRaw := 5;
		END_FOR
		FOR i := 1 TO 3 DO
			gaTemps[i].stTempRead.iRaw := 5;
		END_FOR
		gConductivity.stConductivity.iRaw := 5;
		gFlow.stFlowRate.iRaw := 5;
		UUT();
		tbTBLog := CONCAT(tbTBLog, 'S');
		iTestStep := 2;
	2:
		tbTBLog := CONCAT(tbTBLog, '2');
		FOR i := 1 TO 2 DO
			IF gaPumps[i].stDescription.xFault = TRUE OR gaPumps[i].stDescription.xAlarm = TRUE THEN
				tbTBLog := CONCAT(tbTBLog, 'F');
				iTestStep := 66;
			ELSE
				tbTBLog := CONCAT(tbTBLog, 'S');
				iTestStep := 3;
			END_IF
		END_FOR

	3:
		tbTBLog := CONCAT(tbTBLog, '3');
		FOR i := 1 TO 3 DO
			IF gaTemps[i].stDescription.xFault = TRUE OR gaTemps[i].stDescription.xAlarm = TRUE THEN
				tbTBLog := CONCAT(tbTBLog, 'F');
				iTestStep := 66;
			ELSE
				tbTBLog := CONCAT(tbTBLog, 'S');
				iTestStep := 4;
			END_IF
		END_FOR
	4:
		tbTBLog := CONCAT(tbTBLog, '4');
		IF gConductivity.stDescription.xFault = TRUE OR gConductivity.stDescription.xAlarm = TRUE THEN
				tbTBLog := CONCAT(tbTBLog, 'F');
				iTestStep := 66;
		ELSE
				tbTBLog := CONCAT(tbTBLog, 'S');
				iTestStep := 5;
		END_IF
	5:
		tbTBLog := CONCAT(tbTBLog, '5');
		IF gFlow.stDescription.xFault = TRUE OR gFlow.stDescription.xAlarm = TRUE THEN
				tbTBLog := CONCAT(tbTBLog, 'F ');
				iTestStep := 66;
		ELSE
				tbTBLog := CONCAT(tbTBLog, 'S');
				iTestStep := 6;
		END_IF
	6: (*Pumps should Fault + Alarm*)
		resetVars();
		tbTBLog := CONCAT(tbTBLog, '6');
		gaPumps[1].stPumpPower.iRaw := 3;
		gaPumps[2].stPumpPower.iRaw := 3;
		FOR i := 1 TO 3 DO
			gaTemps[i].stTempRead.iRaw := 5;
		END_FOR
		gConductivity.stConductivity.iRaw := 5;
		gFlow.stFlowRate.iRaw := 5;
		UUT();
		tbTBLog := CONCAT(tbTBLog, 'S');
		iTestStep := 7;
	7:
		tbTBLog := CONCAT(tbTBLog, '7');
		FOR i := 1 TO 2 DO
		IF gaPumps[i].stDescription.xFault = FALSE OR gaPumps[i].stDescription.xAlarm = FALSE THEN
				tbTBLog := CONCAT(tbTBLog, 'F');
				iTestStep := 66;
			ELSE
				tbTBLog := CONCAT(tbTBLog, 'S');
				iTestStep := 8;
			END_IF
		END_FOR

	8:
		tbTBLog := CONCAT(tbTBLog, '8');
		FOR i := 1 TO 3 DO
			IF gaTemps[i].stDescription.xFault = TRUE OR gaTemps[i].stDescription.xAlarm = TRUE THEN
				tbTBLog := CONCAT(tbTBLog, 'F');
				iTestStep := 66;
			ELSE
				tbTBLog := CONCAT(tbTBLog, 'S');
				iTestStep := 9;
			END_IF
		END_FOR
	9:
		tbTBLog := CONCAT(tbTBLog, '9');
		IF gConductivity.stDescription.xFault = TRUE OR gConductivity.stDescription.xAlarm = TRUE THEN
				tbTBLog := CONCAT(tbTBLog, 'F');
				iTestStep := 66;
		ELSE
				tbTBLog := CONCAT(tbTBLog, 'S');
				iTestStep := 10;
		END_IF
	10:
		tbTBLog := CONCAT(tbTBLog, '10');
		IF gFlow.stDescription.xFault = TRUE OR gFlow.stDescription.xAlarm = TRUE THEN
				tbTBLog := CONCAT(tbTBLog, 'F ');
				iTestStep := 66;
		ELSE
				tbTBLog := CONCAT(tbTBLog, 'S');
				iTestStep := 11;
		END_IF
	11: (*Pumps Should Fault*)
		resetVars();
		tbTBLog := CONCAT(tbTBLog, '11');
		gaPumps[1].stPumpPower.iRaw := 30;
		gaPumps[2].stPumpPower.iRaw := 30;
		FOR i := 1 TO 3 DO
			gaTemps[i].stTempRead.iRaw := 5;
		END_FOR
		gConductivity.stConductivity.iRaw := 5;
		gFlow.stFlowRate.iRaw := 5;
		UUT();
		tbTBLog := CONCAT(tbTBLog, 'S');
		iTestStep := iTestStep + 1;
	12:
		tbTBLog := CONCAT(tbTBLog, '12');
		FOR i := 1 TO 2 DO
			IF gaPumps[i].stDescription.xFault = FALSE OR gaPumps[i].stDescription.xAlarm = FALSE THEN
				tbTBLog := CONCAT(tbTBLog, 'F');
				iTestStep := 66;
			ELSE
				tbTBLog := CONCAT(tbTBLog, 'S');
				iTestStep := iTestStep + 1;
			END_IF
		END_FOR

	13:
		tbTBLog := CONCAT(tbTBLog, '13');
		FOR i := 1 TO 3 DO
			IF gaTemps[i].stDescription.xFault = TRUE OR gaTemps[i].stDescription.xAlarm = TRUE THEN
				tbTBLog := CONCAT(tbTBLog, 'F');
				iTestStep := 66;
			ELSE
				tbTBLog := CONCAT(tbTBLog, 'S');
				iTestStep := iTestStep + 1;
			END_IF
		END_FOR
	14:
		tbTBLog := CONCAT(tbTBLog, '14');
		IF gConductivity.stDescription.xFault = TRUE OR gConductivity.stDescription.xAlarm = TRUE THEN
				tbTBLog := CONCAT(tbTBLog, 'F');
				iTestStep := 66;
		ELSE
				tbTBLog := CONCAT(tbTBLog, 'S');
				iTestStep := iTestStep + 1;
		END_IF
	15:
		tbTBLog := CONCAT(tbTBLog, '15');
		IF gFlow.stDescription.xFault = TRUE OR gFlow.stDescription.xAlarm = TRUE THEN
				tbTBLog := CONCAT(tbTBLog, 'F ');
				iTestStep := 66;
		ELSE
				tbTBLog := CONCAT(tbTBLog, 'S');
				iTestStep := iTestStep + 1;
		END_IF
	16: (*Minimum Test - Temps should Fault*)
		resetVars();
		tbTBLog := CONCAT(tbTBLog, INT_TO_STRING(iTestStep));
		gaPumps[1].stPumpPower.iRaw := 5;
		gaPumps[2].stPumpPower.iRaw := 5;
		gaTemps[1].stTempRead.iRaw := 2;
		gaTemps[2].stTempRead.iRaw := 2;
		gaTemps[3].stTempRead.iRaw := 2;
		gConductivity.stConductivity.iRaw := 5;
		gFlow.stFlowRate.iRaw := 5;
		UUT();
		tbTBLog := CONCAT(tbTBLog, 'S');
		iTestStep := iTestStep + 1;
	17:
		tbTBLog := CONCAT(tbTBLog, INT_TO_STRING(iTestStep));
		FOR i := 1 TO 2 DO
			IF gaPumps[i].stDescription.xFault = TRUE OR gaPumps[i].stDescription.xAlarm = TRUE THEN
				tbTBLog := CONCAT(tbTBLog, 'F');
				iTestStep := 66;
			ELSE
				tbTBLog := CONCAT(tbTBLog, 'S');
				iTestStep := iTestStep + 1;
			END_IF
		END_FOR

	18:
		tbTBLog := CONCAT(tbTBLog, INT_TO_STRING(iTestStep));
		FOR i := 1 TO 3 DO
			IF gaTemps[i].stDescription.xFault = FALSE OR gaTemps[i].stDescription.xAlarm = FALSE THEN
				tbTBLog := CONCAT(tbTBLog, 'F');
				iTestStep := 66;
			ELSE
				tbTBLog := CONCAT(tbTBLog, 'S');
				iTestStep := iTestStep + 1;
			END_IF
		END_FOR
	19:
		tbTBLog := CONCAT(tbTBLog, INT_TO_STRING(iTestStep));
		IF gConductivity.stDescription.xFault = TRUE OR gConductivity.stDescription.xAlarm = TRUE THEN
				tbTBLog := CONCAT(tbTBLog, 'F');
				iTestStep := 66;
		ELSE
				tbTBLog := CONCAT(tbTBLog, 'S');
				iTestStep := iTestStep + 1;
		END_IF
	20:
		tbTBLog := CONCAT(tbTBLog, INT_TO_STRING(iTestStep));
		IF gFlow.stDescription.xFault = TRUE OR gFlow.stDescription.xAlarm = TRUE THEN
				tbTBLog := CONCAT(tbTBLog, 'F ');
				iTestStep := 66;
		ELSE
				tbTBLog := CONCAT(tbTBLog, 'S');
				iTestStep := iTestStep + 1;
		END_IF
	21: (*Max Val Test Temp Should Fault*)
		resetVars();
		tbTBLog := CONCAT(tbTBLog, INT_TO_STRING(iTestStep));
		gaPumps[1].stPumpPower.iRaw := 5;
		gaPumps[2].stPumpPower.iRaw := 5;
		gaTemps[i].stTempRead.iRaw := 100;
		gaTemps[2].stTempRead.iRaw := 100;
		gaTemps[3].stTempRead.iRaw := 100;
		gConductivity.stConductivity.iRaw := 5;
		gFlow.stFlowRate.iRaw := 5;
		UUT();
		tbTBLog := CONCAT(tbTBLog, 'S');
		iTestStep := iTestStep + 1;
	22:
		tbTBLog := CONCAT(tbTBLog, INT_TO_STRING(iTestStep));
		FOR i := 1 TO 2 DO
			IF gaPumps[i].stDescription.xFault = TRUE OR gaPumps[i].stDescription.xAlarm = TRUE THEN
				tbTBLog := CONCAT(tbTBLog, 'F');
				iTestStep := 66;
			ELSE
				tbTBLog := CONCAT(tbTBLog, 'S');
				iTestStep := iTestStep + 1;
			END_IF
		END_FOR

	23:
		tbTBLog := CONCAT(tbTBLog, INT_TO_STRING(iTestStep));
		FOR i := 1 TO 3 DO
			IF gaTemps[i].stDescription.xFault = FALSE OR gaTemps[i].stDescription.xAlarm = FALSE THEN
				tbTBLog := CONCAT(tbTBLog, 'F');
				iTestStep := 66;
			ELSE
				tbTBLog := CONCAT(tbTBLog, 'S');
				iTestStep := iTestStep + 1;
			END_IF
		END_FOR
	24:
		tbTBLog := CONCAT(tbTBLog, INT_TO_STRING(iTestStep));
		IF gConductivity.stDescription.xFault = TRUE OR gConductivity.stDescription.xAlarm = TRUE THEN
				tbTBLog := CONCAT(tbTBLog, 'F');
				iTestStep := 66;
		ELSE
				tbTBLog := CONCAT(tbTBLog, 'S');
				iTestStep := iTestStep + 1;
		END_IF
	25:
		tbTBLog := CONCAT(tbTBLog, INT_TO_STRING(iTestStep));
		IF gFlow.stDescription.xFault = TRUE OR gFlow.stDescription.xAlarm = TRUE THEN
				tbTBLog := CONCAT(tbTBLog, 'F ');
				iTestStep := 66;
		ELSE
				tbTBLog := CONCAT(tbTBLog, 'S');
				iTestStep := iTestStep + 1;
		END_IF
	26: (*Min Val Test Cond Should Fault*)
		resetVars();
		tbTBLog := CONCAT(tbTBLog, INT_TO_STRING(iTestStep));
		gaPumps[1].stPumpPower.iRaw := 5;
		gaPumps[2].stPumpPower.iRaw := 5;
		gaTemps[i].stTempRead.iRaw := 5;
		gaTemps[2].stTempRead.iRaw := 5;
		gaTemps[3].stTempRead.iRaw := 5;
		gConductivity.stConductivity.iRaw := 1;
		gFlow.stFlowRate.iRaw := 5;
		UUT();
		tbTBLog := CONCAT(tbTBLog, 'S');
		iTestStep := iTestStep + 1;
	27:
		tbTBLog := CONCAT(tbTBLog, INT_TO_STRING(iTestStep));
		FOR i := 1 TO 2 DO
			IF gaPumps[i].stDescription.xFault = TRUE OR gaPumps[i].stDescription.xAlarm = TRUE THEN
				tbTBLog := CONCAT(tbTBLog, 'F');
				iTestStep := 66;
			ELSE
				tbTBLog := CONCAT(tbTBLog, 'S');
				iTestStep := iTestStep + 1;
			END_IF
		END_FOR

